(* IEC 61131-3 sources: BLM_BACKGROUND/src/PROGRAM_FILES/FC (part 5) *)

		General_State#STATE_END:
			CURRENT_STATE:=GENERAL_STATE#STATE_INIT;

	END_CASE;
	OutputState:=CURRENT_STATE;
END_FUNCTION_BLOCK

FUNCTION Init_Disp

  VAR_EXTERNAL
    Disp                            :ARRAY[(FIRST_DEVICE)..(FIRST_DEVICE+_MAXDEVICES#MAXDEVICES-1)] OF Device;
  END_VAR

  VAR_EXTERNAL CONSTANT
    INTERMEDIATE                    :SINT;
    FIRST_DEVICE                    :INT;
    DISP_IN_V_C :SINT;	//17 - Dispositivo virtuale composto da più dispositivi reali
    DISP_IN_TT  :SINT;		//01 - TEMPO LAVORO - TEMPO RIPOSO   xxxxxxx0001
  END_VAR

  VAR_INPUT
    Ndisp  :INT;
  END_VAR
  Disp[NDisp].Stato:=INTERMEDIATE;
  Disp[NDisp].position:=(DISP[Ndisp].Limite_Lavoro-DISP[Ndisp].Limite_Riposo)/2;
  DISP[NDisp].In_Movimento:=FALSE;
  AbilitazioneDispositivi(Dispositivo:=NDisp, Stato:=TRUE);
 (* {
  #ifdef EMULAZIONE_INPUT
  }*)
		IF Disp[NDisp].TipoIn<>DISP_IN_V_C THEN
			Disp[NDisp].TipoIn:=DISP_IN_TT;
    END_IF;
	(*{
  #endif  //Fine EMULAZIONE_INPUT
  }*)
END_FUNCTION

FUNCTION AbilitazioneDispositivi

  VAR_EXTERNAL
    Disp                            :ARRAY[(FIRST_DEVICE)..(FIRST_DEVICE+_MAXDEVICES#MAXDEVICES-1)] OF Device;
  END_VAR

  VAR_EXTERNAL CONSTANT
    FIRST_DEVICE                    :INT;
  END_VAR

  VAR_INPUT
    Dispositivo    :INT;
    Stato      :BOOL;
  END_VAR
  Disp[Dispositivo].consenso_minus:=Stato;
  Disp[Dispositivo].consenso_plus:=Stato;
END_FUNCTION

FUNCTION StartTimerRisparmioEnergetico

  VAR_EXTERNAL
    MinuteSavingEnergy              :INT;
    StatusStandBy                   :BOOL;
    TimerSistema                :ARRAY[0..MAX_TIMER_SISTEMA-1] OF Timer;
  END_VAR

  VAR_EXTERNAL CONSTANT
    T_ENERGY_SAVING    	            :INT;
    MAX_TIMER_SISTEMA 	            :USINT;
  END_VAR

  VAR_INPUT
    Tempo  :INT;
  END_VAR;
  IF MinuteSavingEnergy>0 THEN
    StatusStandBy:=FALSE;
    TimerSistema[T_ENERGY_SAVING].Value:=Tempo*60000.0;
    TimerSistema[T_ENERGY_SAVING].Status:=SINT#1;
  END_IF;
END_FUNCTION

FUNCTION ReadDigitalInput:BOOL

  VAR_EXTERNAL
    SystemStarted                   :BOOL;
    IAddress                        : ARRAY [0..MAXDIGITALINPUT] OF Digital_Input;
    O_EmergencyFromSimotion		      :BOOL;	//Only to be able to compile machines without safety PLCs
    InputWithoutAddress             :DINT;
    i_sys_DpCoupler                 :BOOL;
    i_sys_PnCoupler                 :BOOL;
    i_sys_StatusIOoptional          :BOOL;
    i_sys_StatusIOAL42               :BOOL;
    i_sys_StatusIOAL5                :BOOL;
    i_sys_StatusIOAL5Optional       :BOOL;
  END_VAR

  VAR_EXTERNAL CONSTANT
    MAXDIGITALINPUT                    :INT;
    INP_OUT_TIPO_SAFETY					       :SINT;
    INP_EMERGENCY                      :INT;
    ERR_IO_NOT_DEFINED                 :DINT ; //Manca associazione virtuale/fisico
  END_VAR

  VAR_INPUT
    NumInput  :DINT;
    Verifica  :BOOL:=FALSE;
  END_VAR

  VAR
    Porta     :DINT;
    Bit       :USINT;
    iret      :INT;
    OldStato  :BOOL;
  END_VAR

  IF NumInput>=0 AND SystemStarted=TRUE THEN
    IF IAddress[NumInput].Enable_Forzatura=TRUE THEN
      (*{
      #ifdef EMULAZIONE
			}*)
				IF IAddress[NumInput].Stato_Forzatura=FALSE THEN
					ReadDigitalInput:=FALSE;
				ELSE
					ReadDigitalInput:=TRUE;
				END_IF;
      (*{
      #else  //Fine EMULAZIONE
      }*)
				IF IAddress[NumInput].Port=INP_OUT_TIPO_SAFETY OR IAddress[NumInput].Bit=INP_OUT_TIPO_SAFETY THEN
					//Gli ingressi il cui stato è impostato dal plc di sicurezza non si possono forzare, tranne
					//l^ingresso di emergenza che può essere forzato solo basso (per esigenze di teleassistenza).
					IF NumInput=INP_EMERGENCY AND IAddress[NumInput].Enable_Forzatura=TRUE THEN
						IAddress[NumInput].Stato_Forzatura:=FALSE;
						ReadDigitalInput:=FALSE;
						O_EmergencyFromSimotion:=TRUE;
					ELSE
          	IAddress[NumInput].Enable_Forzatura:=FALSE;
					END_IF;
        ELSE
					//Ingressi standard si possono forzare
          IF IAddress[NumInput].STATO_FORZATURA=FALSE THEN
            ReadDigitalInput:=FALSE;
          ELSE
            ReadDigitalInput:=TRUE;
          END_IF;
        END_IF;
      (*{
      #endif  //Fine NO EMULAZIONE
      }*)
    ELSE
      Porta:=IAddress[NumInput].Port;
      Bit:=TO_USINT(IAddress[NumInput].Bit);
      IF IAddress[NumInput].Port=INP_OUT_TIPO_SAFETY AND IAddress[NumInput].Bit=INP_OUT_TIPO_SAFETY THEN
        //Lettura dello stato degli ingressi che vengono valorizzati da informazioni proveniente dal plc di sicurezza
        ReadDigitalInput:=LetturaIngressiSafety(NumeroInput:=NumInput);
      ELSE
        //Lettura ingressi collegati ai moduli standard e non impostati dal plc di sicurezza
        IF Verifica=TRUE AND (Porta<0 OR Bit<0) THEN
          //Verifica, se necessario, la definizione del collegamento virtuale fisico
          InputWithoutAddress:=NumInput;
          iret:=Push_error(Code:=ERR_IO_NOT_DEFINED, Arresto:=FALSE);
          ReadDigitalInput:=FALSE;
        ELSE
          OldStato:=FALSE;
          ReadDigitalInput:=LetturaIngressiDpCoupler(OldStato:=OldStato,
                                                     UsoDpCoupler:=i_sys_DpCoupler,
                                                     Porta:=porta,
                                                     Bit:=bit);
          OldStato:=ReadDigitalInput;
          ReadDigitalInput:=LetturaIngressiPnCoupler(OldStato:=OldStato,
                                                     UsoPnCoupler:=i_sys_PnCoupler,
                                                     Porta:=porta,
                                                     Bit:=bit);
          OldStato:=ReadDigitalInput;
          ReadDigitalInput:=LetturaIngressiSiemensProfinet(OldStato:=OldStato,
                                                           Porta:=porta,
                                                           Bit:=bit);
          OldStato:=ReadDigitalInput;
          ReadDigitalInput:=LetturaIngressiSiemensProfibus(OldStato:=OldStato,
                                                           Porta:=porta,
                                                           Bit:=bit,
                                                           StatoIOopzionale:=i_sys_StatusIOoptional,
                                                           StatoIOAL42:=i_sys_StatusIOAL42,
                                                           StatoIOAL5:=i_sys_StatusIOAL5,
                                                           StatoIOAL5Opzionale:=i_sys_StatusIOAL5Optional);
          OldStato:=ReadDigitalInput;
          ReadDigitalInput:=LetturaIngressiFestoProfinet(OldStato:=OldStato,
                                                         Porta:=porta,
                                                         Bit:=bit);
        END_IF;
      END_IF;
      IF IAddress[NumInput].inversione=TRUE THEN
        ///Inversione dello stato dell^ingresso fisico se prevista la proprietà
        IF ReadDigitalInput=TRUE THEN
          ReadDigitalInput:=FALSE;
        ELSE
          ReadDigitalInput:=TRUE;
        END_IF;
      END_IF;
    END_IF;  //Fine else degli ingressi di tipo standard port>-1 bit>-1
  ELSE
    ReadDigitalInput:=FALSE;
  END_IF;
END_FUNCTION

/**************************************************
 * READING STATUS OF VALUED INPUTS VIA SAFETY PLC *
 **************************************************/

FUNCTION LetturaIngressiSafety:BOOL

  VAR_EXTERNAL
    I_Emergenza,
    I_Barriera,
    I_RiarmoAzionamenti,
    I_Barriera_2,
    I_Pedale,
    I_Hold_To_Run,
    I_Radar_Zona_1,
    I_Radar_Zona_2,
    I_Radar_Zona_3,
    //Stato degli ingressi dei moduli di sicurezza
        //Stato degli ingressi dei moduli di sicurezza
    I_Modulo_1_Input_1,I_Modulo_1_Input_2,I_Modulo_1_Input_3,I_Modulo_1_Input_4,
    I_Modulo_2_Input_1,I_Modulo_2_Input_2,I_Modulo_2_Input_3,I_Modulo_2_Input_4,
    I_Modulo_3_Input_1,I_Modulo_3_Input_2,I_Modulo_3_Input_3,I_Modulo_3_Input_4  : BOOL;
  END_VAR

  VAR_EXTERNAL CONSTANT
    INP_PHOTOCELLS_NOT_VIOLATED             :INT;
    INP_MEASURE_TERMINAL_TUBE               :INT;
    INP_SEARCH_WELD                         :INT;
    INP_INTEGRATED_SOUL                     :INT;
    INP_EMERGENCY                           :INT;
    INP_RESET_DRIVES                        :INT;
    INP_BARRIER_2                           :INT;
    INP_PEDALE_SAFETY                       :INT;
    INP_HOLD_TO_RUN                         :INT;
    INP_EMERGENCY_PLC_SAFETY						    :INT;
    INP_PHOTOCELLS_NOT_VIOLATED_PLC_SAFETY	:INT;
    INP_HOLD_TO_RUN_PLC_SAFETY						  :INT;
    INP_PEDALE_SAFETY_PLC_SAFETY					  :INT;
    INP_RESET_DRIVE_PLC_SAFETY				      :INT;
    INP_BARRIER_2_PLC_SAFETY						    :INT;
    INP_OPTICAL_REARMING_PLC_SAFETY					:INT;
    INP_BARRIERA_3_PLC_SAFETY						    :INT;
    INP_EMERGENCY_EXTERIOR_PLC_SAFETY				:INT;
    INP_EXTERNAL_BARRIER_PLC_SAFETY					:INT;
    INP_RESET_EXTERNAL_DRIVES_PLC_SAFETY	  :INT;
    INP_RADAR_ZONA_BIT_0_PLC_SAFETY					:INT;
    INP_RADAR_ZONA_BIT_1_PLC_SAFETY					:INT;
    INP_RADAR_ZONA_1                        :INT;
    INP_RADAR_ZONA_2                        :INT;
    INP_RADAR_ZONA_3                        :INT;
    INP_RADAR_ZONA_BIT_0                    :INT;
    INP_RADAR_ZONA_BIT_1                    :INT;

  END_VAR

  VAR_INPUT
    MeasuringInput         : DB_ANY;
    NumeroInput  :DINT;
  END_VAR

  VAR
    Weld_Marker : REF_TO TO_MeasuringInput;
  END_VAR

  CASE NumeroInput OF
    (*{
    #ifdef SAFETY_INTEGRATED
    }
      INP_SAFETY_UOMO_MORTO:
        LetturaIngressiSafety:=i_sys_UomoMorto;
    {
    #endif  //Fine SAFETY_INTEGRATED
    }*)
    (*{
    #ifdef ORBITALE
    }
      {
      #ifdef FOTOCELLULA_MISURA_X1 %%%%
      }*)
        // INP_MEASURE_TERMINAL_TUBE:
        //   IF _to.FotocellulaMisuraX1.actualinputstate=POSITIVE THEN
        //     LetturaIngressiSafety:=TRUE;
        //   ELSE
        //     LetturaIngressiSafety:=FALSE;
        //   END_IF;
      (*{
      #endif  //Fine FOTOCELLULA_MISURA_X1
      }
    {
    #else  //Fine ORBITALE
    }*)
      INP_SEARCH_WELD, INP_INTEGRATED_SOUL:
        //Nelle macchine prima serie si usava lo stesso ingresso fisico
        //per leggere due diversi dispositivi
        Weld_Marker:= AsMeasuringInputRef(MeasuringInput);
        IF Weld_Marker^.InputState = TRUE THEN
          LetturaIngressiSafety:=TRUE;
        ELSE
          LetturaIngressiSafety:=FALSE;
        END_IF;
    (*{
    #endif  //Fine NO ORBITALE
    }
    {
    #ifdef PROFINET
    }*)
      INP_EMERGENCY:
        LetturaIngressiSafety:=I_Emergenza;
      INP_PHOTOCELLS_NOT_VIOLATED:
        LetturaIngressiSafety:=I_Barriera;
        INP_RESET_DRIVES:
        LetturaIngressiSafety:=I_RiarmoAzionamenti;
      INP_BARRIER_2:
        LetturaIngressiSafety:=I_Barriera_2;
			(*{
      #ifndef ORBITALE
      }*)
        INP_PEDALE_SAFETY:
          LetturaIngressiSafety:=I_Pedale;
        INP_HOLD_TO_RUN:
          LetturaIngressiSafety:=I_Hold_To_Run;
      (*{
      #endif  //Fine NO ORBITALE
      }
			{
			#ifdef DIAGNOSTICA_PLC_SAFETY
			}*)
				//Ingressi di diagnosdtica per visualizzazione in BlmMotion
				INP_EMERGENCY_PLC_SAFETY:
					LetturaIngressiSafety:=I_Modulo_1_Input_1;
        INP_PHOTOCELLS_NOT_VIOLATED_PLC_SAFETY:
					LetturaIngressiSafety:=I_Modulo_1_Input_2;
				(*{
				#ifndef ORBITALE
				}*)
					INP_HOLD_TO_RUN_PLC_SAFETY:
						LetturaIngressiSafety:=I_Modulo_1_Input_3;
					INP_PEDALE_SAFETY_PLC_SAFETY:
						LetturaIngressiSafety:=I_Modulo_2_Input_1;
				(*{
				#endif	//Fine NO ORBITALE
				}*)
				INP_RESET_DRIVE_PLC_SAFETY:
					LetturaIngressiSafety:=I_Modulo_1_Input_4;
				(*{
				#ifdef PLC_S7_1500
				}*)
					//Nuovo hardware associato a Tia portal
					INP_BARRIER_2_PLC_SAFETY:
						LetturaIngressiSafety:=I_Modulo_2_Input_2;
          INP_OPTICAL_REARMING_PLC_SAFETY	:
						LetturaIngressiSafety:=I_Modulo_2_Input_3;
					INP_BARRIERA_3_PLC_SAFETY:
						LetturaIngressiSafety:=I_Modulo_2_Input_4;
          INP_EMERGENCY_EXTERIOR_PLC_SAFETY:
						LetturaIngressiSafety:=I_Modulo_3_Input_1;
          INP_EXTERNAL_BARRIER_PLC_SAFETY:
						LetturaIngressiSafety:=I_Modulo_3_Input_2;
          INP_RESET_EXTERNAL_DRIVES_PLC_SAFETY:
						LetturaIngressiSafety:=I_Modulo_3_Input_3;
				(*{
				#else //FINE PLC_S7_1500
				}*)
					//Vecchio hardware associato a Step7
					(*{
					#ifdef ORBITALE
					}
            INP_BARRIER_2_PLC_SAFETY:
							(*{
							#ifdef DH4010
							}
								LetturaIngressiSafety:=I_Modulo_2_Input_2;
							(*{
							#else	//Fine DH4010
							}
								LetturaIngressiSafety:=I_Modulo_1_Input_3;
							(*{
							#endif	//Fine NO DH4010
							}
					{
					#else	//Fine ORBITALE
					}
            INP_BARRIER_2_PLC_SAFETY:
							LetturaIngressiSafety:=I_Modulo_2_Input_2;*)
						INP_RADAR_ZONA_BIT_0_PLC_SAFETY:
							LetturaIngressiSafety:=I_Modulo_2_Input_3;
						INP_RADAR_ZONA_BIT_1_PLC_SAFETY:
							LetturaIngressiSafety:=I_Modulo_2_Input_4;
						//Con la selezione a 3 bit di 3 zone radar l^impostazione
						//degli ingressi che vengono realmente cablati al PLC safety è:
						//0 0 1 = Zona 1
						//0 1 0 = Zona 2
						//1 0 0 = Zona 3
						INP_RADAR_ZONA_1:
							LetturaIngressiSafety:=I_Radar_Zona_1;
						INP_RADAR_ZONA_2:
							LetturaIngressiSafety:=I_Radar_Zona_2;
						INP_RADAR_ZONA_3:
							LetturaIngressiSafety:=I_Radar_Zona_3;
						//Con la selezione a 2 bit di 3 zone l^impostazione
						//degli ingressi che vengono realmente cablati al PLC safety è:
						//1 0 = Zona 1
						//0 1 = Zona 2
						//0 0 = Zona 3
						INP_RADAR_ZONA_BIT_0:
							IF I_Radar_Zona_1=TRUE THEN
								LetturaIngressiSafety:=FALSE;
							END_IF;
							IF I_Radar_Zona_2=TRUE THEN
								LetturaIngressiSafety:=TRUE;
							END_IF;
							IF I_Radar_Zona_3=TRUE THEN
								LetturaIngressiSafety:=FALSE;
							END_IF;
						INP_RADAR_ZONA_BIT_1:
							IF I_Radar_Zona_1=TRUE THEN
								LetturaIngressiSafety:=TRUE;
							END_IF;
							IF I_Radar_Zona_2=TRUE THEN
								LetturaIngressiSafety:=FALSE;
							END_IF;
							IF I_Radar_Zona_3=TRUE THEN
								LetturaIngressiSafety:=FALSE;
							END_IF;
					(*{
					#endif	//Fine NO ORBITALE
					}
				{
				#endif //FINE NO PLC_S7_1500
				}
			{
			#endif	//Fine DIAGNOSTICA_PLC_SAFETY
			}
    {
    #endif  //Fine PROFINET
    } *)
  END_CASE;
END_FUNCTION

FUNCTION LetturaIngressiDpCoupler:BOOL

  VAR_EXTERNAL
    V_dbcoupler_i  : dbcoupler_i;
  END_VAR

  VAR_INPUT
    OldStato      :BOOL;
    UsoDpCoupler  :BOOL;
    Porta					:DINT;
    Bit						:USINT;
  END_VAR

    LetturaIngressiDpCoupler:=OldStato;
    IF UsoDpCoupler=TRUE THEN
      CASE porta OF
      //Ingressi da DpCoupler
      900:LetturaIngressiDpCoupler:=getbit(V_dbcoupler_i.address_db_i[0], bit);//dbcoupler_i00.%X0; //_getbit(dbcoupler_i00, bit);
      901:LetturaIngressiDpCoupler:=getbit(V_dbcoupler_i.address_db_i[1], bit);
      902:LetturaIngressiDpCoupler:=getbit(V_dbcoupler_i.address_db_i[2], bit);
      903:LetturaIngressiDpCoupler:=getbit(V_dbcoupler_i.address_db_i[3], bit);
      904:LetturaIngressiDpCoupler:=getbit(V_dbcoupler_i.address_db_i[4], bit);
      905:LetturaIngressiDpCoupler:=getbit(V_dbcoupler_i.address_db_i[5], bit);
      906:LetturaIngressiDpCoupler:=getbit(V_dbcoupler_i.address_db_i[6], bit);
      907:LetturaIngressiDpCoupler:=getbit(V_dbcoupler_i.address_db_i[7], bit);
      908:LetturaIngressiDpCoupler:=getbit(V_dbcoupler_i.address_db_i[8], bit);
      909:LetturaIngressiDpCoupler:=getbit(V_dbcoupler_i.address_db_i[9], bit);
      910:LetturaIngressiDpCoupler:=getbit(V_dbcoupler_i.address_db_i[10], bit);
      911:LetturaIngressiDpCoupler:=getbit(V_dbcoupler_i.address_db_i[11], bit);
      912:LetturaIngressiDpCoupler:=getbit(V_dbcoupler_i.address_db_i[12], bit);
      913:LetturaIngressiDpCoupler:=getbit(V_dbcoupler_i.address_db_i[13], bit);
      914:LetturaIngressiDpCoupler:=getbit(V_dbcoupler_i.address_db_i[14], bit);
      915:LetturaIngressiDpCoupler:=getbit(V_dbcoupler_i.address_db_i[15], bit);
      916:LetturaIngressiDpCoupler:=getbit(V_dbcoupler_i.address_db_i[16], bit);
      917:LetturaIngressiDpCoupler:=getbit(V_dbcoupler_i.address_db_i[17], bit);
      918:LetturaIngressiDpCoupler:=getbit(V_dbcoupler_i.address_db_i[18], bit);
      919:LetturaIngressiDpCoupler:=getbit(V_dbcoupler_i.address_db_i[19], bit);
      920:LetturaIngressiDpCoupler:=getbit(V_dbcoupler_i.address_db_i[20], bit);
      921:LetturaIngressiDpCoupler:=getbit(V_dbcoupler_i.address_db_i[21], bit);
      922:LetturaIngressiDpCoupler:=getbit(V_dbcoupler_i.address_db_i[22], bit);
      923:LetturaIngressiDpCoupler:=getbit(V_dbcoupler_i.address_db_i[23], bit);
      924:LetturaIngressiDpCoupler:=getbit(V_dbcoupler_i.address_db_i[24], bit);
      925:LetturaIngressiDpCoupler:=getbit(V_dbcoupler_i.address_db_i[25], bit);
      926:LetturaIngressiDpCoupler:=getbit(V_dbcoupler_i.address_db_i[26], bit);
      927:LetturaIngressiDpCoupler:=getbit(V_dbcoupler_i.address_db_i[27], bit);
      928:LetturaIngressiDpCoupler:=getbit(V_dbcoupler_i.address_db_i[28], bit);
      929:LetturaIngressiDpCoupler:=getbit(V_dbcoupler_i.address_db_i[29], bit);
      930:LetturaIngressiDpCoupler:=getbit(V_dbcoupler_i.address_db_i[30], bit);
      931:LetturaIngressiDpCoupler:=getbit(V_dbcoupler_i.address_db_i[31], bit);
      932:LetturaIngressiDpCoupler:=getbit(V_dbcoupler_i.address_db_i[32], bit);
      933:LetturaIngressiDpCoupler:=getbit(V_dbcoupler_i.address_db_i[33], bit);
      934:LetturaIngressiDpCoupler:=getbit(V_dbcoupler_i.address_db_i[34], bit);
      935:LetturaIngressiDpCoupler:=getbit(V_dbcoupler_i.address_db_i[35], bit);
      936:LetturaIngressiDpCoupler:=getbit(V_dbcoupler_i.address_db_i[36], bit);
      937:LetturaIngressiDpCoupler:=getbit(V_dbcoupler_i.address_db_i[37], bit);
      938:LetturaIngressiDpCoupler:=getbit(V_dbcoupler_i.address_db_i[38], bit);
      939:LetturaIngressiDpCoupler:=getbit(V_dbcoupler_i.address_db_i[39], bit);
      940:LetturaIngressiDpCoupler:=getbit(V_dbcoupler_i.address_db_i[40], bit);
      941:LetturaIngressiDpCoupler:=getbit(V_dbcoupler_i.address_db_i[41], bit);
      942:LetturaIngressiDpCoupler:=getbit(V_dbcoupler_i.address_db_i[42], bit);
      943:LetturaIngressiDpCoupler:=getbit(V_dbcoupler_i.address_db_i[43], bit);
      944:LetturaIngressiDpCoupler:=getbit(V_dbcoupler_i.address_db_i[44], bit);
      945:LetturaIngressiDpCoupler:=getbit(V_dbcoupler_i.address_db_i[45], bit);
      946:LetturaIngressiDpCoupler:=getbit(V_dbcoupler_i.address_db_i[46], bit);
      947:LetturaIngressiDpCoupler:=getbit(V_dbcoupler_i.address_db_i[47], bit);
      948:LetturaIngressiDpCoupler:=getbit(V_dbcoupler_i.address_db_i[48], bit);
      949:LetturaIngressiDpCoupler:=getbit(V_dbcoupler_i.address_db_i[49], bit);
      950:LetturaIngressiDpCoupler:=getbit(V_dbcoupler_i.address_db_i[50], bit);
      951:LetturaIngressiDpCoupler:=getbit(V_dbcoupler_i.address_db_i[51], bit);
      952:LetturaIngressiDpCoupler:=getbit(V_dbcoupler_i.address_db_i[52], bit);
      953:LetturaIngressiDpCoupler:=getbit(V_dbcoupler_i.address_db_i[53], bit);
      954:LetturaIngressiDpCoupler:=getbit(V_dbcoupler_i.address_db_i[54], bit);
      955:LetturaIngressiDpCoupler:=getbit(V_dbcoupler_i.address_db_i[55], bit);
      956:LetturaIngressiDpCoupler:=getbit(V_dbcoupler_i.address_db_i[56], bit);
      957:LetturaIngressiDpCoupler:=getbit(V_dbcoupler_i.address_db_i[57], bit);
      958:LetturaIngressiDpCoupler:=getbit(V_dbcoupler_i.address_db_i[58], bit);
      959:LetturaIngressiDpCoupler:=getbit(V_dbcoupler_i.address_db_i[59], bit);
      960:LetturaIngressiDpCoupler:=getbit(V_dbcoupler_i.address_db_i[60], bit);
      961:LetturaIngressiDpCoupler:=getbit(V_dbcoupler_i.address_db_i[61], bit);
      962:LetturaIngressiDpCoupler:=getbit(V_dbcoupler_i.address_db_i[62], bit);
      963:LetturaIngressiDpCoupler:=getbit(V_dbcoupler_i.address_db_i[63], bit);
    END_CASE;
  END_IF;
END_FUNCTION

/***********************************************************************
 * READING STATUS OF VALUED INPUTS VIA PNPNCOUPLER ON PROFINET NETWORK *
 ***********************************************************************/

 FUNCTION LetturaIngressiPnCoupler:BOOL

  VAR_EXTERNAL
    V_pncoupler_i  : pncoupler_i;

  END_VAR

  VAR_INPUT
    OldStato      :BOOL;
    UsoPnCoupler	:BOOL;
    Porta					:DINT;
    Bit						:USINT;
  END_VAR
  LetturaIngressiPnCoupler:=OldStato;
  {::ifdef PROFINET}
    IF UsoPnCoupler=TRUE THEN
      CASE porta OF
        //Ingressi da PnCoupler
        900:LetturaIngressiPnCoupler:=getbit(V_pncoupler_i.address_pn_i[0], bit);
        901:LetturaIngressiPnCoupler:=getbit(V_pncoupler_i.address_pn_i[1], bit);
        902:LetturaIngressiPnCoupler:=getbit(V_pncoupler_i.address_pn_i[2], bit);
        903:LetturaIngressiPnCoupler:=getbit(V_pncoupler_i.address_pn_i[3], bit);
        904:LetturaIngressiPnCoupler:=getbit(V_pncoupler_i.address_pn_i[4], bit);
        905:LetturaIngressiPnCoupler:=getbit(V_pncoupler_i.address_pn_i[5], bit);
        906:LetturaIngressiPnCoupler:=getbit(V_pncoupler_i.address_pn_i[6], bit);
        907:LetturaIngressiPnCoupler:=getbit(V_pncoupler_i.address_pn_i[7], bit);
        908:LetturaIngressiPnCoupler:=getbit(V_pncoupler_i.address_pn_i[8], bit);
        909:LetturaIngressiPnCoupler:=getbit(V_pncoupler_i.address_pn_i[9], bit);
        910:LetturaIngressiPnCoupler:=getbit(V_pncoupler_i.address_pn_i[10], bit);
        911:LetturaIngressiPnCoupler:=getbit(V_pncoupler_i.address_pn_i[11], bit);
        912:LetturaIngressiPnCoupler:=getbit(V_pncoupler_i.address_pn_i[12], bit);
        913:LetturaIngressiPnCoupler:=getbit(V_pncoupler_i.address_pn_i[13], bit);
        914:LetturaIngressiPnCoupler:=getbit(V_pncoupler_i.address_pn_i[14], bit);
        915:LetturaIngressiPnCoupler:=getbit(V_pncoupler_i.address_pn_i[15], bit);
        916:LetturaIngressiPnCoupler:=getbit(V_pncoupler_i.address_pn_i[16], bit);
        917:LetturaIngressiPnCoupler:=getbit(V_pncoupler_i.address_pn_i[17], bit);
        918:LetturaIngressiPnCoupler:=getbit(V_pncoupler_i.address_pn_i[18], bit);
        919:LetturaIngressiPnCoupler:=getbit(V_pncoupler_i.address_pn_i[19], bit);
        920:LetturaIngressiPnCoupler:=getbit(V_pncoupler_i.address_pn_i[20], bit);
        921:LetturaIngressiPnCoupler:=getbit(V_pncoupler_i.address_pn_i[21], bit);
        922:LetturaIngressiPnCoupler:=getbit(V_pncoupler_i.address_pn_i[22], bit);
        923:LetturaIngressiPnCoupler:=getbit(V_pncoupler_i.address_pn_i[23], bit);
        924:LetturaIngressiPnCoupler:=getbit(V_pncoupler_i.address_pn_i[23], bit);
        925:LetturaIngressiPnCoupler:=getbit(V_pncoupler_i.address_pn_i[25], bit);
        926:LetturaIngressiPnCoupler:=getbit(V_pncoupler_i.address_pn_i[26], bit);
        927:LetturaIngressiPnCoupler:=getbit(V_pncoupler_i.address_pn_i[27], bit);
        928:LetturaIngressiPnCoupler:=getbit(V_pncoupler_i.address_pn_i[28], bit);
        929:LetturaIngressiPnCoupler:=getbit(V_pncoupler_i.address_pn_i[29], bit);
        930:LetturaIngressiPnCoupler:=getbit(V_pncoupler_i.address_pn_i[30], bit);
        931:LetturaIngressiPnCoupler:=getbit(V_pncoupler_i.address_pn_i[31], bit);
        932:LetturaIngressiPnCoupler:=getbit(V_pncoupler_i.address_pn_i[32], bit);
        933:LetturaIngressiPnCoupler:=getbit(V_pncoupler_i.address_pn_i[33], bit);
        934:LetturaIngressiPnCoupler:=getbit(V_pncoupler_i.address_pn_i[34], bit);
        935:LetturaIngressiPnCoupler:=getbit(V_pncoupler_i.address_pn_i[35], bit);
        936:LetturaIngressiPnCoupler:=getbit(V_pncoupler_i.address_pn_i[36], bit);
        937:LetturaIngressiPnCoupler:=getbit(V_pncoupler_i.address_pn_i[37], bit);
        938:LetturaIngressiPnCoupler:=getbit(V_pncoupler_i.address_pn_i[38], bit);
        939:LetturaIngressiPnCoupler:=getbit(V_pncoupler_i.address_pn_i[39], bit);
        940:LetturaIngressiPnCoupler:=getbit(V_pncoupler_i.address_pn_i[40], bit);
        941:LetturaIngressiPnCoupler:=getbit(V_pncoupler_i.address_pn_i[41], bit);
        942:LetturaIngressiPnCoupler:=getbit(V_pncoupler_i.address_pn_i[42], bit);
        943:LetturaIngressiPnCoupler:=getbit(V_pncoupler_i.address_pn_i[43], bit);
        944:LetturaIngressiPnCoupler:=getbit(V_pncoupler_i.address_pn_i[44], bit);
        945:LetturaIngressiPnCoupler:=getbit(V_pncoupler_i.address_pn_i[45], bit);
        946:LetturaIngressiPnCoupler:=getbit(V_pncoupler_i.address_pn_i[46], bit);
        947:LetturaIngressiPnCoupler:=getbit(V_pncoupler_i.address_pn_i[47], bit);
        948:LetturaIngressiPnCoupler:=getbit(V_pncoupler_i.address_pn_i[48], bit);
        949:LetturaIngressiPnCoupler:=getbit(V_pncoupler_i.address_pn_i[49], bit);
        950:LetturaIngressiPnCoupler:=getbit(V_pncoupler_i.address_pn_i[50], bit);
        951:LetturaIngressiPnCoupler:=getbit(V_pncoupler_i.address_pn_i[51], bit);
        952:LetturaIngressiPnCoupler:=getbit(V_pncoupler_i.address_pn_i[52], bit);
        953:LetturaIngressiPnCoupler:=getbit(V_pncoupler_i.address_pn_i[53], bit);
        954:LetturaIngressiPnCoupler:=getbit(V_pncoupler_i.address_pn_i[54], bit);
        955:LetturaIngressiPnCoupler:=getbit(V_pncoupler_i.address_pn_i[55], bit);
        956:LetturaIngressiPnCoupler:=getbit(V_pncoupler_i.address_pn_i[56], bit);
        957:LetturaIngressiPnCoupler:=getbit(V_pncoupler_i.address_pn_i[57], bit);
        958:LetturaIngressiPnCoupler:=getbit(V_pncoupler_i.address_pn_i[58], bit);
        959:LetturaIngressiPnCoupler:=getbit(V_pncoupler_i.address_pn_i[59], bit);
        960:LetturaIngressiPnCoupler:=getbit(V_pncoupler_i.address_pn_i[60], bit);
        961:LetturaIngressiPnCoupler:=getbit(V_pncoupler_i.address_pn_i[61], bit);
        962:LetturaIngressiPnCoupler:=getbit(V_pncoupler_i.address_pn_i[62], bit);
        963:LetturaIngressiPnCoupler:=getbit(V_pncoupler_i.address_pn_i[63], bit);
      END_CASE;
    END_IF;
  {::endif}  //Fine PROFINET

END_FUNCTION

FUNCTION LetturaIngressiSiemensProfinet:BOOL

  VAR_EXTERNAL
    i_sys_StatoIOAL5_old			              :BOOL;
    i_sys_StatoIOAL5Opzionale_old           :BOOL;
    i_sys_StatoIOAL5                        :BOOL;
    i_sys_StatoIOAL5Opzionale               :BOOL;
    V_ph_i  : ph_i;
    V_ph_i_old  : ph_i_old;
    V_PHIAL5_Opz  : PHIAL5_Opz;
    V_PHIAL5_Opz_old  : PHIAL5_Opz_old;

                X122_d0 : BOOL;
                X122_d1 : BOOL;
                X122_d2 : BOOL;
                X122_d3 : BOOL;
                X122_d16 : BOOL;
                X122_d17 : BOOL;

                X132_d4 : BOOL;
                X132_d5 : BOOL;
                X132_d6 : BOOL;
                X132_d7 : BOOL;
                X132_d20 : BOOL;
                X132_d21 : BOOL;
  END_VAR

  VAR_EXTERNAL CONSTANT
    INDIRIZZO_X122_SINAMICS             :INT;
    INDIRIZZO_X132_SINAMICS             :INT;
  END_VAR

  VAR_INPUT
    OldStato:BOOL;
    Porta		:DINT;
    Bit			:USINT;
  END_VAR;

  LetturaIngressiSiemensProfinet:=OldStato;
  CASE Porta OF
    //Macchine seconda serie con profinet
    00:LetturaIngressiSiemensProfinet:=getbit(V_ph_i.address_ph_i[0], bit);  //32.0÷7
    01:LetturaIngressiSiemensProfinet:=getbit(V_ph_i.address_ph_i[1], bit);  //33.0÷7
    02:LetturaIngressiSiemensProfinet:=getbit(V_ph_i.address_ph_i[2], bit);  //34.0÷7
    //Ingressi opzionali
    03:LetturaIngressiSiemensProfinet:=getbit(V_ph_i.address_ph_i[3], bit);  //37.0÷7
    04:LetturaIngressiSiemensProfinet:=getbit(V_ph_i.address_ph_i[4], bit);  //38.0÷7
  END_CASE;
  {::ifdef AL_BLM}
    IF i_sys_StatoIOAL5_old=TRUE THEN
      CASE Porta OF
        //IM 151-3 PN ST (STEP 7)ingressi standard AL5
        08:LetturaIngressiSiemensProfinet:=getbit(V_ph_i_old.address_ph_i_old[0], bit);  //42.0÷3
        09:LetturaIngressiSiemensProfinet:=getbit(V_ph_i_old.address_ph_i_old[1], bit);  //43.0÷3
        10:LetturaIngressiSiemensProfinet:=getbit(V_ph_i_old.address_ph_i_old[2], bit);  //44.0÷3
        11:LetturaIngressiSiemensProfinet:=getbit(V_ph_i_old.address_ph_i_old[3], bit);  //45.0÷3
        12:LetturaIngressiSiemensProfinet:=getbit(V_ph_i_old.address_ph_i_old[4], bit);  //46.0÷3
        13:LetturaIngressiSiemensProfinet:=getbit(V_ph_i_old.address_ph_i_old[5], bit);  //47.0÷3
        14:LetturaIngressiSiemensProfinet:=getbit(V_ph_i_old.address_ph_i_old[6], bit);  //48.0÷3
      END_CASE;
    END_IF;
    IF i_sys_StatoIOAL5Opzionale_old=TRUE THEN
      CASE Porta OF
        //IM 151-3 PN ST (STEP 7)ingressi opzionali
        15:LetturaIngressiSiemensProfinet:=getbit(V_PHIAL5_Opz_old.address_PHIAL5_Opz_old[0], bit);  //49.0÷3
        16:LetturaIngressiSiemensProfinet:=getbit(V_PHIAL5_Opz_old.address_PHIAL5_Opz_old[1], bit);  //50.0÷3
        17:LetturaIngressiSiemensProfinet:=getbit(V_PHIAL5_Opz_old.address_PHIAL5_Opz_old[2], bit);  //51.0÷3
        18:LetturaIngressiSiemensProfinet:=getbit(V_PHIAL5_Opz_old.address_PHIAL5_Opz_old[3], bit);  //52.0÷3
        19:LetturaIngressiSiemensProfinet:=getbit(V_PHIAL5_Opz_old.address_PHIAL5_Opz_old[4], bit);  //53.0÷3
        20:LetturaIngressiSiemensProfinet:=getbit(V_PHIAL5_Opz_old.address_PHIAL5_Opz_old[5], bit);  //54.0÷3
        21:LetturaIngressiSiemensProfinet:=getbit(V_PHIAL5_Opz_old.address_PHIAL5_Opz_old[6], bit);  //55.0÷3
      END_CASE;
    END_IF;

    IF i_sys_StatoIOAL5=TRUE THEN
      //IM 155-6 PN HF (TIA PORTAL) ingressi standard AL5
      CASE Porta OF
        05:LetturaIngressiSiemensProfinet:=getbit(V_ph_i_old.address_ph_i_old[0], bit);  //42.0÷7
        06:LetturaIngressiSiemensProfinet:=getbit(V_ph_i_old.address_ph_i_old[1], bit);  //43.0÷7
        07:LetturaIngressiSiemensProfinet:=getbit(V_ph_i_old.address_ph_i_old[2], bit);  //44.0÷7
        08:LetturaIngressiSiemensProfinet:=getbit(V_ph_i_old.address_ph_i_old[3], bit);  //45.0÷7
      END_CASE;
    END_IF;
    IF i_sys_StatoIOAL5Opzionale THEN
      //IM 155-6 PN HF (TIA PORTAL) ingressi opzionali
      CASE Porta OF
        12:LetturaIngressiSiemensProfinet:=getbit(V_PHIAL5_Opz.address_PHIAL5_Opz[0], bit);  //49.0÷7
        13:LetturaIngressiSiemensProfinet:=getbit(V_PHIAL5_Opz.address_PHIAL5_Opz[1], bit);  //50.0÷7
        14:LetturaIngressiSiemensProfinet:=getbit(V_PHIAL5_Opz.address_PHIAL5_Opz[2], bit);  //51.0÷7
        15:LetturaIngressiSiemensProfinet:=getbit(V_PHIAL5_Opz.address_PHIAL5_Opz[3], bit);  //52.0÷7
      END_CASE;
    END_IF;
  {::endif}  //Fine AL_BLM

  // CASE Porta OF
    // {::ifdef TAVOLI_ELETTRICI} %%%%

    //   23:LetturaIngressiSiemensProfinet:=getbit(I_Tavoli_0, bit);
    //   24:LetturaIngressiSiemensProfinet:=getbit(I_Tavoli_1, bit);
    //   25:LetturaIngressiSiemensProfinet:=getbit(I_Tavoli_2, bit);
    // {::endif} //FINE TAVOLI ELETTRICI

      {::ifndef EMULAZIONE}

      INDIRIZZO_X122_SINAMICS:
        CASE bit OF
          0:LetturaIngressiSiemensProfinet:=X122_d0;
          1:LetturaIngressiSiemensProfinet:=X122_d1;
          2:LetturaIngressiSiemensProfinet:=X122_d2;
          3:LetturaIngressiSiemensProfinet:=X122_d3;
          8:LetturaIngressiSiemensProfinet:=X122_d16;
          9:LetturaIngressiSiemensProfinet:=X122_d17;
        END_CASE;

      INDIRIZZO_X132_SINAMICS:
        CASE bit OF
          0:LetturaIngressiSiemensProfinet:=X132_d4;
          1:LetturaIngressiSiemensProfinet:=X132_d5;
          2:LetturaIngressiSiemensProfinet:=X132_d6;
          3:LetturaIngressiSiemensProfinet:=X132_d7;
          8:LetturaIngressiSiemensProfinet:=X132_d20;
          9:LetturaIngressiSiemensProfinet:=X132_d21;
        END_CASE;
      {::endif}  //Fine NO EMULAZIONE

  // END_CASE;

END_FUNCTION
// {
// #else //FINE PLC_S7_1500
// }

/**************************************************************************
 * READING STATUS OF INPUTS VALUED BY SIEMENS MODULES ON PROFIBUS NETWORK *
 **************************************************************************/

FUNCTION LetturaIngressiSiemensProfibus:BOOL

  VAR_EXTERNAL
    X122_d0 : BOOL;
    X122_d1 : BOOL;
    X122_d2 : BOOL;
    X122_d3 : BOOL;

    X132_d4 : BOOL;
    X132_d5 : BOOL;
    X132_d6 : BOOL;
    X132_d7 : BOOL;

    V_ph_i                   : ph_i;
    V_PHIAL5_Opz             : PHIAL5_Opz;

    // PHIAL5_Opz_1  :BYTE;
    // PHIAL5_Opz_2 :BYTE;
    // PHIAL5_Opz_3 :BYTE;
    // PHIAL5_Opz_4 :BYTE;
    // PHIAL5_Opz_5  :BYTE;
    // PHIAL5_Opz_6 :BYTE;
    // PHIAL5_Opz_7  :BYTE;

    // phi00  :BYTE;
    // phi01  :BYTE;
    // phi02  :BYTE;
    // phi03  :BYTE;
    // phi04  :BYTE;
  END_VAR

  VAR_EXTERNAL CONSTANT
    INDIRIZZO_X122_SINAMICS             :INT;
    INDIRIZZO_X132_SINAMICS             :INT;
  END_VAR

  VAR_INPUT
    OldStato            :BOOL;
    Porta								:DINT;
    Bit									:USINT;
    StatoIOopzionale    :BOOL;
    StatoIOAL42					:BOOL;
    StatoIOAL5          :BOOL;
    StatoIOAL5Opzionale	:BOOL;
  END_VAR

  LetturaIngressiSiemensProfibus:=OldStato;
  //{::ifndef PROFINET}%%%%
    // IF StatoIOopzionale=TRUE THEN %%%%
      //Modulo IO opzionale
    //   CASE porta OF
    //     00:LetturaIngressiSiemensProfibus:=getbit(PHI00_opzionale,bit);
    //     01:LetturaIngressiSiemensProfibus:=getbit(PHI01_opzionale,bit);
    //     02:LetturaIngressiSiemensProfibus:=getbit(PHI02_opzionale,bit);
    //     03:LetturaIngressiSiemensProfibus:=getbit(PHI03_opzionale,bit);
    //     04:LetturaIngressiSiemensProfibus:=getbit(PHI04_opzionale,bit);
    //     08:LetturaIngressiSiemensProfibus:=getbit(PHI08_opzionale,bit);
    //     09:LetturaIngressiSiemensProfibus:=getbit(PHI09_opzionale,bit);
    //     10:LetturaIngressiSiemensProfibus:=getbit(PHI10_opzionale,bit);
    //   END_CASE;
    // ELSE
    //   //Modulo IO standard
    //   CASE porta OF
    //     00:LetturaIngressiSiemensProfibus:=getbit(PHI00,bit);
    //     01:LetturaIngressiSiemensProfibus:=getbit(PHI01,bit);
    //     02:LetturaIngressiSiemensProfibus:=getbit(PHI02,bit);
    //     03:LetturaIngressiSiemensProfibus:=getbit(PHI03,bit);
    //     04:LetturaIngressiSiemensProfibus:=getbit(PHI04,bit);
    //   END_CASE;
    // END_IF;
    {::ifndef EMULAZIONE}
      CASE porta OF
        INDIRIZZO_X122_SINAMICS:
          CASE bit OF
            0:LetturaIngressiSiemensProfibus:=X122_d0;
            1:LetturaIngressiSiemensProfibus:=X122_d1;
            2:LetturaIngressiSiemensProfibus:=X122_d2;
            3:LetturaIngressiSiemensProfibus:=X122_d3;
          END_CASE;
        INDIRIZZO_X132_SINAMICS:
          CASE bit OF
            0:LetturaIngressiSiemensProfibus:=X132_d4;
            1:LetturaIngressiSiemensProfibus:=X132_d5;
            2:LetturaIngressiSiemensProfibus:=X132_d6;
            3:LetturaIngressiSiemensProfibus:=X132_d7;
          END_CASE;
      END_CASE;
    {::endif}  //Fine NO EMULAZIONE
    {::ifdef AL_BLM}
    //   {
    //   #ifdef ETURN %%%%
    //   }
        // IF StatoIOAL42=TRUE THEN
        //   CASE porta OF
        //     11:LetturaIngressiSiemensProfibus:=getbit(PHI20,bit);
        //     12:LetturaIngressiSiemensProfibus:=getbit(PHI21,bit);
        //     13:LetturaIngressiSiemensProfibus:=getbit(PHI22,bit);
        //     14:LetturaIngressiSiemensProfibus:=getbit(PHI23,bit);
        //     15:LetturaIngressiSiemensProfibus:=getbit(PHI24,bit);
        //   END_CASE;
        // END_IF;
      // {
      // #endif  //Fine ETURN
      // }
      // IF StatoIOAL5=TRUE THEN
      //   CASE porta OF
      //     11:LetturaIngressiSiemensProfibus:=getbit(PHI20_opzionale, bit);
      //     12:LetturaIngressiSiemensProfibus:=getbit(PHI21_opzionale, bit);
      //     13:LetturaIngressiSiemensProfibus:=getbit(PHI22_opzionale, bit);
      //     14:LetturaIngressiSiemensProfibus:=getbit(PHI23_opzionale, bit);
      //     15:LetturaIngressiSiemensProfibus:=getbit(PHI24_opzionale, bit);
      //     16:LetturaIngressiSiemensProfibus:=getbit(PHI25_opzionale, bit);
      //     17:LetturaIngressiSiemensProfibus:=getbit(PHI26_opzionale, bit);
      //   END_CASE;
      // END_IF;
      // {::ifdef MODULO_ROLAND} %%%%
      //   IF StatoIOAL5Opzionale=TRUE THEN
      //     CASE porta OF
      //       18:LetturaIngressiSiemensProfibus:=getbit(PHIAL5_Opz_1, bit);
      //       19:LetturaIngressiSiemensProfibus:=getbit(PHIAL5_Opz_2, bit);
      //       20:LetturaIngressiSiemensProfibus:=getbit(PHIAL5_Opz_3, bit);
      //       21:LetturaIngressiSiemensProfibus:=getbit(PHIAL5_Opz_4, bit);
      //       22:LetturaIngressiSiemensProfibus:=getbit(PHIAL5_Opz_5, bit);
      //       23:LetturaIngressiSiemensProfibus:=getbit(PHIAL5_Opz_6, bit);
      //       24:LetturaIngressiSiemensProfibus:=getbit(PHIAL5_Opz_7, bit);
      //     END_CASE;
      //   END_IF;
      // {::endif}  //Fine MODULO_ROLAND

  {::endif}  //Fine AL_BLM

  // {
  // #endif  //Fine NO PROFINET
  // }
END_FUNCTION

/**************************************************************************
 * READING STATUS OF INPUTS VALUED BY SIEMENS MODULES ON PROFIBUS NETWORK *
 **************************************************************************/

FUNCTION LetturaIngressiFestoProfinet:BOOL

  VAR_EXTERNAL CONSTANT
    FESTO_INP_LINEA_1_MODULO_1          :INT;  //bit 0÷15  16 input
    FESTO_INP_LINEA_1_MODULO_3          :INT;  //bit 0÷07  08 input
    FESTO_INP_LINEA_2_MODULO_2          :INT;  //bit 0÷15  16 input
    FESTO_INP_LINEA_2_MODULO_3          :INT;  //bit 0÷07  08 input
    FESTO_INP_LINEA_3_MODULO_2          :INT;  //bit 0÷15  16 input
    FESTO_INP_LINEA_3_MODULO_3          :INT;  //bit 0÷07  08 input
    FESTO_INP_LINEA_4_MODULO_2          :INT;  //bit 0÷15  16 input
    FESTO_INP_LINEA_4_MODULO_3          :INT;  //bit 0÷07  08 input
END_VAR

  VAR_INPUT
    OldStato	:BOOL;
    Porta			:DINT;
    Bit				:USINT;
  END_VAR
  LetturaIngressiFestoProfinet:=OldStato;
  {::ifdef IO_FESTO_PROFINET}
    CASE porta OF
      FESTO_INP_LINEA_1_MODULO_1:
        LetturaIngressiFestoProfinet:=getbit(festo_inp_linea_1a, bit);  //16 ingressi
      FESTO_INP_LINEA_1_MODULO_3:
        LetturaIngressiFestoProfinet:=getbit(festo_inp_linea_1b, bit);  //08 ingressi
      FESTO_INP_LINEA_2_MODULO_2:
        LetturaIngressiFestoProfinet:=getbit(festo_inp_linea_2a, bit);  //16 ingressi
      FESTO_INP_LINEA_2_MODULO_3:
        LetturaIngressiFestoProfinet:=getbit(festo_inp_linea_2b, bit);  //08 ingressi
      FESTO_INP_LINEA_3_MODULO_2:
        LetturaIngressiFestoProfinet:=getbit(festo_inp_linea_3a, bit);  //16 ingressi
      FESTO_INP_LINEA_3_MODULO_3:
        LetturaIngressiFestoProfinet:=getbit(festo_inp_linea_3b, bit);  //08 ingressi
      FESTO_INP_LINEA_4_MODULO_2:
        LetturaIngressiFestoProfinet:=getbit(festo_inp_linea_4a, bit);  //16 ingressi
      FESTO_INP_LINEA_4_MODULO_3:
        LetturaIngressiFestoProfinet:=getbit(festo_inp_linea_4b, bit);  //08 ingressi
    END_CASE;
  {::endif} //Fine IO_FESTO_PROFINET

  ;

END_FUNCTION

FUNCTION_BLOCK FB_EnableMasterAxisBLM

  VAR_EXTERNAL
    AssiMaster                      :ARRAY[FIRST_AXIS_MASTER..FIRST_AXIS_MASTER+_CONST_VAR_DEF._MAXAXIS_MASTER#MAXAXIS_MASTER-1] OF MasterAxis;
  END_VAR

  VAR_EXTERNAL CONSTANT

    FIRST_AXIS_MASTER				        :INT;

  END_VAR

	VAR_INPUT
		NumMaster	:INT;
		//Asse			:PosAxis;
	END_VAR

	VAR
		dret					:LREAL;
		CURRENT_STATE	:INT;
		//thisCommand		:CommandIDType;
	END_VAR

	VAR_OUTPUT
		OutputState:INT;
	END_VAR
	CASE CURRENT_STATE OF
		GENERAL_STATE#STATE_INIT:
			(*IF UsoPLCOpen THEN
				//PLCOpen*)
				AssiMaster[NumMaster].MC_Axes.enable_axes :=TRUE;
				CURRENT_STATE:=GENERAL_STATE#STATE_END;
			(*ELSE
				thisCommand:=_getCommandID();
				CURRENT_STATE:=STATE_ENABLEMASTER_ENABLE;
			END_IF;

		STATE_ENABLEMASTER_ENABLE:
			dret:=_enableAxis(axis:=Asse,
							movingMode:=POSITION_CONTROLLED,
							enableMode:=ALL,
							servoControlMode:=ACTIVE,
							servoCommandToActualMode:=INACTIVE,
							nextCommand:=IMMEDIATELY,
							commandId:=thisCommand,
							forcecontrolMode:=INACTIVE);
			IF (ModoAttesa=WHEN_COMMAND_DONE) THEN
				IF (dret<>7001 AND dret<>7002) THEN
					CURRENT_STATE:=STATE_END;
				END_IF;
			ELSE*)
				CURRENT_STATE:=GENERAL_STATE#STATE_END;
			//END_IF;

		GENERAL_STATE#STATE_END:
			CURRENT_STATE:=GENERAL_STATE#STATE_INIT;
	END_CASE;
	OutputState:=CURRENT_STATE;
END_FUNCTION_BLOCK

/**********************************************************************
 * RESET OF OUTPUTS THAT NEED TO BE RESET WITH CYCLE STOP AND STORAGE *
 *                     OF THE STATE BEFORE RESET                      *
 **********************************************************************/
FUNCTION OnStopCicloDispositivi

  VAR_EXTERNAL
    OAddress                        : ARRAY [0..MAXDIGITALOUTPUT] OF Digital_Output;
  END_VAR

  VAR_EXTERNAL CONSTANT
    MAXDIGITALOUTPUT                    :INT;
    MAXDIGITALINPUT                     :INT;
  END_VAR

  VAR
    i    :DINT;
  END_VAR;
  FOR i:=0 TO MAXDIGITALOUTPUT DO
    IF oaddress[i].AbilGestStopCiclo=TRUE THEN
			IF oaddress[i].stato=TRUE THEN
				//Si memorizza lo stato dell^uscita solamente se è attiva
				oaddress[i].statoprestopciclo:=oaddress[i].stato;
			END_IF;
      WriteDigitalOutput(NumOutput:=i, Value:=FALSE);
    END_IF;
  END_FOR;
END_FUNCTION

/*****************************************************************************
 * READS FROM THE STATE TABLE THE VALUE INDICATED BY THE ROW AND COLUMN. THE *
 *                 PROGRAMME NUMBER FROM 0 TO MAXPROGRAMS-1                  *
 *****************************************************************************/

FUNCTION ReadTabStati:REAL

  VAR_EXTERNAL
    Programmi                      :ARRAY[0.._CONST_VAR_DEF._MPROGRAMS#MAXPROGRAMS - UINT#1] OF Programma;
    // {
    // #ifdef DH4010
    // }
    TabellaStati	:ARRAY[TABLE#TABLE_LX ..TABLE#TABLE_RX ] OF TabStato;
  END_VAR

  VAR_EXTERNAL CONSTANT
    ERR_NUMSTATES                       :DINT;
  END_VAR

  VAR_INPUT
    Riga,
    Colonna,
    Programma	:INT;
    Tabella   :SINT;
  END_VAR

  VAR
    Puntatore	:DINT;
    iret      :INT;
  END_VAR

  ;
//  {
//   #ifdef DH4010
//   }
    // IF GetNumberOfStates(Tabella:=Tabella, Programma:=Programma)>0 THEN
    //   Puntatore:=Riga+Programmi[Programma].TabStatiInizio[Tabella];
    //   ReadTabStati:=TabellaStati[Tabella][Puntatore][Colonna];
    // ELSE
    //   iret:=Push_error(Code:=ERR_NUMSTATES, Arresto:=FALSE, Attesa:=FALSE);
    // END_IF;
  // {
  // #else  //Fine DH4010
  // }
    // IF GetNumberOfStates(Tabella:=Tabella, Programma:=Programma)>0 THEN
    //   Puntatore:=Riga+Programmi[Programma].TabStatiInizio;
    //   ReadTabStati:=TabellaStati[Puntatore][Colonna];
    // ELSE
    //   iret:=Push_error(Code:=ERR_NUMSTATES, Arresto:=FALSE, Attesa:=FALSE);
    // END_IF;
  // {
  // #endif  //Fine NO DH4010
  // }
END_FUNCTION

FUNCTION SetAxSwLimit1

  VAR_EXTERNAL
    pm                              : ARRAY[_FIRST_AXIS#FIRST_AXIS.._FIRST_AXIS#FIRST_AXIS+_CONST_VAR_DEF._MAXIS#MAXAXIS-1] OF AxisParameters;
  END_VAR

  VAR_EXTERNAL CONSTANT
    EXTRALIMIT         	:REAL ; // extralimite per limiti fisici
    Q1 : INT;
    V1 : INT;
  END_VAR

  VAR_INPUT
		PrimoAsseNoGestione		:INT:=-1;
		SecondoAsseNoGestione	:INT:=-1;
		TerzoAsseNoGestione		:INT:=-1;
		QuartoAsseNoGestione	:INT:=-1;
		QuintoAsseNoGestione	:INT:=-1;
		SestoAsseNoGestione		:INT:=-1;
  END_VAR
  VAR
    i											:INT;
		Eseguire							:BOOL:=TRUE;
  END_VAR
  FOR i:=_FIRST_AXIS#FIRST_AXIS TO _FIRST_AXIS#FIRST_AXIS+_MAXIS#MAXAXIS-1 DO
    pm[i].MA_LIMITE_ATTIVO:=1;
    IF i<>PrimoAsseNoGestione AND i<>SecondoAsseNoGestione AND
       i<>TerzoAsseNoGestione AND i<>QuartoAsseNoGestione AND
       i<>QuintoAsseNoGestione AND i<>SestoAsseNoGestione THEN
			(*{
			#ifdef ELECTXL
			}*)
				IF i=Q1 OR i=V1 THEN
					//Per ELECT-XL occorre gestire i limiti degli assi Q1 e V1 quando è abilitato da VGP
					//l^accessorio
					Eseguire:=Set_Limiti_Q1V1()=FALSE ;
				END_IF;
			(*{
			#endif //Fine ELECTXL
			}*)
			IF Eseguire=TRUE THEN
				//Se non sono in monitoring attivo i limiti software 1 agli assi, considerando la posizione
				//attuale del^asse
				ImpostaLimiteSW(Asse:=i, ValoreMinus:=pm[i].Ma_Pos_Limit_Minus_Attivo-EXTRALIMIT);
				ImpostaLimiteSW(Asse:=i, ValorePlus:=pm[i].Ma_Pos_Limit_Plus_Attivo+EXTRALIMIT);
			END_IF;
    END_IF;
  END_FOR;
END_FUNCTION

/**********************************************************************************************************************
 *           WITH ACCESSORY MO00003632 (INCREASE AXIS TRAVEL Q1 FOR MEDIUM RADIUS UP TO 610MM, THE TRAVELS            *
 *                                   OF Q1 AND V1 ACCORDING TO THE FOLLOWING RULES:                                   *
 *      - MAXIMUM LIMIT INCREASE OF Q1, INDICATED BY VGP VIA THE VARIABLE CFG.LIMQ1CAUSATODAV1, IF THE POSITION       *
 *              OF V1 IS HIGHER THAN THE POSITION INDICATED BY VGP IN THE VARIABLE CFG.LIMV1CAUSATODAQ1               *
 *      - RECORDING OF THE STANDARD POSITIVE LIMIT OF Q1, INDICATED IN PARAMETER M36110, WHEN THE POSITION OF V1      *
 *                   IS LOWER THAN THE VALUE INDICATED BY VGP IN THE VARIABLE CFG.LIMV1CAUSATODAQ1                    *
 * - REDUCTION OF THE NEGATIVE LIMIT OF V1 TO THE VALUE INDICATED BY VGP IN THE VARIABLE CFG.LIMV1CAUSATODAQ1, IF THE *
 *           POSITION OF Q1 IS HIGHER THAN THE STANDARD POSITIVE LIMIT INDICATED IN THE PARAMETER IN M36110           *
 *   - REDETERMINATION OF THE STANDARD NEGATIVE LIMIT OF V1, INDICATED IN PARAMETER M36110, WHEN THE POSITION OF Q1   *
 *                         IS LOWER THAN THE POSITIVE LIMIT OF Q1 GIVEN IN PARAMETER M36110.                          *
 **********************************************************************************************************************/

 (*{
#ifdef ELECTXL
}*)
	FUNCTION Set_Limiti_Q1V1:BOOL

    VAR_EXTERNAL
    cfg                             :_TYPE.Config_Struct;
    pm                              : ARRAY[_FIRST_AXIS#FIRST_AXIS.._FIRST_AXIS#FIRST_AXIS+_CONST_VAR_DEF._MAXIS#MAXAXIS-1] OF AxisParameters;
    Axes                            :ARRAY[_FIRST_AXIS#FIRST_AXIS.._FIRST_AXIS#FIRST_AXIS+_CONST_VAR_DEF._MAXIS#MAXAXIS-1] OF ax;/// ax as structure is defined in _TYPE
  END_VAR

    VAR_EXTERNAL CONSTANT
      EXTRALIMIT         	                :REAL; // extralimite per limiti fisici
      MY_BIG_VALUE_REAL                   :REAL;
      V1 : INT;
      Q1 : INT;
    END_VAR

    VAR
      PosAx : REF_TO TO_SynchronousAxis;
    END_VAR

		IF cfg.LimQ1CausatoDaV1<MY_BIG_VALUE_REAL-1 AND cfg.LimQ1CausatoDaV1<>-1 AND
			 cfg.LimV1CausatoDaQ1<MY_BIG_VALUE_REAL-1 AND cfg.LimV1CausatoDaQ1<>-1 THEN
			//Gestione limite V1 in funzione della posizione di Q1
      PosAx := AsSynchronousAxisRef(Axes[Q1].PosAx);
			IF PosAx^.ActualPosition>pm[Q1].Ma_Pos_Limit_Plus THEN
				ImpostaLimiteSw(Asse:=V1, ValoreMinus:=cfg.LimV1CausatoDaQ1-EXTRALIMIT);
			ELSE
				ImpostaLimiteSw(Asse:=V1, ValoreMinus:=pm[V1].Ma_Pos_Limit_Minus-EXTRALIMIT);
			END_IF;
			//Gestione limite Q1 in funzione della posizione di V1
      PosAx := AsSynchronousAxisRef(Axes[V1].PosAx);
			IF PosAx^.ActualPosition>cfg.LimV1CausatoDaQ1 THEN
				ImpostaLimiteSw(Asse:=Q1, ValorePlus:=cfg.LimQ1CausatoDaV1+EXTRALIMIT);
			ELSE
				ImpostaLimiteSw(Asse:=Q1, ValorePlus:=pm[Q1].Ma_Pos_Limit_Plus+EXTRALIMIT);
			END_IF;
			Set_Limiti_Q1V1:=TRUE;
		ELSE
			Set_Limiti_Q1V1:=FALSE;
		END_IF;
	END_FUNCTION
(*{
#endif //FINE ELECTXL
}*)

/****************************************************
 * TRUE IF THE INDICATED AXLE IS READY FOR MOVEMENT *
 ****************************************************/

FUNCTION TestAssePronto:BOOL

  VAR_EXTERNAL
    Axes                            :ARRAY[_FIRST_AXIS#FIRST_AXIS.._FIRST_AXIS#FIRST_AXIS+_CONST_VAR_DEF._MAXIS#MAXAXIS-1] OF ax;/// ax as structure is defined in _TYPE
  END_VAR

  VAR_INPUT
    Asse  :INT;
  END_VAR
  ;
  // IF  CheckIfTOactive(Axis:=Asse)=TRUE THEN %%%%%
  //   IF Axes[Asse].PosAx.actormonitoring.drivestate=ACTIVE AND
  //      Axes[Asse].PosAx.actormonitoring.power=ACTIVE THEN
  //     TestAssePronto:=TRUE;
  //   ELSE
  //     TestAssePronto:=FALSE;
  //   END_IF;
  // END_IF;
END_FUNCTION

/*******************************************************************
 * REACTIVATION OF OUTPUTS WHICH MUST BE RESET WITH CYCLE STOP AND *
 *     SUBSEQUENTLY RESET WITH THE VALUE MEMORISED WITH START      *
 *******************************************************************/

FUNCTION OffStopCicloDispositivi

  VAR_EXTERNAL
    i_sys_stopcond      : INT; // 0=NO STOP, 1=STOP ATTIVO
  END_VAR

  VAR_EXTERNAL CONSTANT
    MAXDIGITALOUTPUT                    :INT;
    OAddress                        : ARRAY [0..MAXDIGITALOUTPUT] OF Digital_Output;
  END_VAR
  VAR
    i    :DINT;
  END_VAR;
  FOR i:=0 TO MAXDIGITALOUTPUT DO
    IF oaddress[i].AbilGestStopCiclo=TRUE AND
       i_sys_stopcond=0 AND
       oaddress[i].StatoPreStopCiclo=TRUE THEN
      WriteDigitalOutput(NumOutput:=i, Value:=oaddress[i].statoprestopciclo);
      oaddress[i].statoprestopciclo:=FALSE;
    END_IF;
  END_FOR;
END_FUNCTION

FUNCTION ResetAllOutStopPoint

  VAR_EXTERNAL CONSTANT
    PRIMO_STOP_POINT_SET_OUT              	:INT;
    MAX_INP_OUT_STOP_POINT                  :INT;
    PRIMO_STOP_POINT_RESET_OUT            	:INT; //252
    ULTIMO_STOP_POINT_SET_OUT             	:INT;//251
    ULTIMO_STOP_POINT_RESET_OUT           	:INT;//275
  END_VAR

  VAR
    i :INT;
  END_VAR
  FOR i:=PRIMO_STOP_POINT_RESET_OUT TO ULTIMO_STOP_POINT_RESET_OUT DO
    OutStopPoint(Codice:=i, Stato:=FALSE);
  END_FOR;
END_FUNCTION

/*************************************
 * SETTING COMMAND OUTPUTS FROM STOP *
 *************************************/
FUNCTION OutStopPoint

  VAR_EXTERNAL CONSTANT
    PRIMO_STOP_POINT_SET_OUT              	:INT;
    MAX_INP_OUT_STOP_POINT                  :INT;
    PRIMO_STOP_POINT_RESET_OUT            	:INT; //252
    ULTIMO_STOP_POINT_SET_OUT             	:INT;//251
    ULTIMO_STOP_POINT_RESET_OUT           	:INT;//275
    ADDRES_OUT_STOPP: ARRAY[PRIMO_STOP_POINT_SET_OUT..ULTIMO_STOP_POINT_SET_OUT] OF INT;
  END_VAR

  VAR_INPUT
    Codice  :LREAL;
    Stato   :BOOL;
  END_VAR
  VAR
    i       :INT;
    dret    :DINT;
  END_VAR
  IF Stato=TRUE THEN
    FOR i:=PRIMO_STOP_POINT_SET_OUT TO ULTIMO_STOP_POINT_SET_OUT DO
      IF Codice=i THEN
        WriteDigitalOutput(NumOutput:=ADDRES_OUT_STOPP[TO_INT(Codice)], Value:=Stato);
      END_IF;
    END_FOR;
  ELSE
    FOR i:=PRIMO_STOP_POINT_RESET_OUT TO ULTIMO_STOP_POINT_RESET_OUT DO
      IF Codice=i THEN
        WriteDigitalOutput(NumOutput:=ADDRES_OUT_STOPP[TO_INT(Codice-MAX_INP_OUT_STOP_POINT)], Value:=Stato);
      END_IF;
    END_FOR;
  END_IF;
END_FUNCTION

FUNCTION Set_Disp

  VAR_EXTERNAL
    Disp                            :ARRAY[(FIRST_DEVICE)..(FIRST_DEVICE+_MAXDEVICES#MAXDEVICES-1)] OF Device;
    OAddress                        : ARRAY [0..MAXDIGITALOUTPUT] OF Digital_Output;
    MinutiRisparmioEnergetico       :INT;
  END_VAR

  VAR_EXTERNAL CONSTANT
    FIRST_DEVICE                          :INT;
    MAXDIGITALOUTPUT                      :INT;
    DISP_IN_TT                            :SINT;		//01 - TEMPO LAVORO - TEMPO RIPOSO   xxxxxxx0001
    DISP_IN_TM                            :SINT;		//03 - TEMPO LAVORO - MICRO RIPOSO   xxxxxxx0011
    DISP_IN_MT                            :SINT;		//05 - MICRO LAVORO - TEMPO RIPOSO   xxxxxxx0101
    DISP_IN_MM                            :SINT;		//07 - MICRO LAVORO - MICRO RIPOSO   xxxxxxx0111
    DISP_IN_AI	                          :SINT;		//09 - INGRESSO ANALOGICO      xxxxxxx1001
    DISP_IN_V                             :SINT;	//16 - INGRESSO VIRTUALE       xxxxxx10000 COMANDATO DALLA LOGICA INTERNA (es: un altro task)

    DISP_OUT_DO                           :SINT;		//1 - USCITA DIGITALE         xxxxxxxxx01
    DISP_OUT_AO                           :SINT; 	//3 - USCITA ANALOGICA        xxxxxxxxx11

  END_VAR

  VAR_INPUT
    Ndisp            :INT;
    Stato            :INT;
    TimerRisparmio  :BOOL;
  END_VAR
  VAR
    Valore          :REAL;
    dret            :DINT;
  END_VAR
  Disp[Ndisp].StatoRichiesto:=Stato;
  IF Disp[NDisp].Enable=FALSE THEN ;
    oaddress[Ndisp].stato:=FALSE;
    // GOTO End;
  END_IF;
  IF TimerRisparmio=TRUE THEN
    StartTimerRisparmioEnergetico(Tempo:=MinutiRisparmioEnergetico);
  END_IF;
  CASE Disp[Ndisp].TipoOut OF
    DISP_OUT_DO:
      IF Disp[Ndisp].spegnimentouscita=TRUE THEN
        IF Disp[Ndisp].Stato=Disp[Ndisp].StatoRichiesto THEN ;
          // GOTO End;
        END_IF;
      END_IF;
      IF Stato=DEVICES_STATUS#LAVORO THEN
        WriteDigitalOutput(NumOutput:=DISP[Ndisp].Out_Riposo, Value:=FALSE);
        WriteDigitalOutput(NumOutput:=DISP[Ndisp].Out_Riposo_2, Value:=FALSE);
        IF DISP[Ndisp].Ritardo_Uscite>0 THEN
          WriteDigitalOutput(NumOutput:=DISP[Ndisp].Out_Lavoro, Value:=TRUE);
          //dret:=_waitTime(timeValue:=REAL_TO_TIME(DISP[Ndisp].Ritardo_Uscite*1000));
          WriteDigitalOutput(NumOutput:=DISP[Ndisp].Out_Lavoro_2, Value:=TRUE);
        ELSE
          WriteDigitalOutput(NumOutput:=DISP[Ndisp].Out_Lavoro_2, Value:=TRUE);
          //dret:=_waitTime(timeValue:=REAL_TO_TIME(ABS(DISP[Ndisp].Ritardo_Uscite*1000)));
          WriteDigitalOutput(NumOutput:=DISP[Ndisp].Out_Lavoro, Value:=TRUE);
        END_IF;
      ELSE
        IF Stato=DEVICES_STATUS#RIPOSO THEN
          WriteDigitalOutput(NumOutput:=DISP[Ndisp].Out_Lavoro, Value:=FALSE);
          WriteDigitalOutput(NumOutput:=DISP[Ndisp].Out_Lavoro_2, Value:=FALSE);
          WriteDigitalOutput(NumOutput:=DISP[Ndisp].Out_Riposo, Value:=TRUE);
          WriteDigitalOutput(NumOutput:=DISP[Ndisp].Out_Riposo_2, Value:=TRUE);
        END_IF;
      END_IF;
    DISP_OUT_AO:;
      //Uscita analogica
  END_CASE;
  //Muove solo se non si trova già sullo stato finale
  IF Stato<>DISP[Ndisp].Stato THEN
    //Doppia uscita digitale
    CASE DISP[Ndisp].TipoIn OF
      DISP_IN_TT:
        //Tempo lavoro, Tempo riposo
        IF Stato=DEVICES_STATUS#LAVORO THEN
          IF Disp[NDisp].Stato<>DEVICES_STATUS#VERSO_LAVORO OR NOT DISP[NDisp].In_Movimento THEN
            DISP[NDisp].Timer:=((DISP[Ndisp].limite_Lavoro-DISP[Ndisp].Position)/DISP[Ndisp].Vel_Lavoro*1000);
          END_IF;
          Disp[NDisp].Stato:=DEVICES_STATUS#VERSO_LAVORO;
          DISP[NDisp].In_Movimento:=TRUE;
        ELSE
          IF Stato=DEVICES_STATUS#RIPOSO THEN
            IF Disp[NDisp].Stato<>DEVICES_STATUS#VERSO_RIPOSO OR NOT DISP[NDisp].In_Movimento THEN
              DISP[NDisp].Timer:=(DISP[Ndisp].Position-DISP[Ndisp].Limite_Riposo)/DISP[Ndisp].Vel_Riposo*1000;
            END_IF;
            Disp[NDisp].Stato:=DEVICES_STATUS#VERSO_RIPOSO;
            DISP[NDisp].In_Movimento:=TRUE;
          END_IF;
        END_IF;
      DISP_IN_TM:  // 3  - TEMPO LAVORO - MICRO RIPOSO   xxxxxxx0011
        IF Stato=DEVICES_STATUS#LAVORO THEN
          IF Disp[NDisp].Stato<>DEVICES_STATUS#VERSO_LAVORO OR NOT DISP[NDisp].In_Movimento THEN
            DISP[NDisp].Timer:=((DISP[Ndisp].Limite_Lavoro-DISP[Ndisp].Position)/DISP[Ndisp].Vel_Lavoro*1000);
          END_IF;
          Disp[NDisp].Stato:=DEVICES_STATUS#VERSO_LAVORO;
          DISP[NDisp].In_Movimento:=TRUE;
        ELSE
          IF Stato=DEVICES_STATUS#RIPOSO THEN
            IF Disp[NDisp].Stato<>DEVICES_STATUS#VERSO_RIPOSO OR NOT DISP[NDisp].In_Movimento THEN
              DISP[NDisp].Timer:=((DISP[Ndisp].Position-DISP[Ndisp].Limite_Riposo)/DISP[Ndisp].Vel_Lavoro*1000);
            END_IF;
            DISP[NDisp].In_Movimento:=TRUE;
            Disp[NDisp].Stato:=DEVICES_STATUS#VERSO_RIPOSO;
          END_IF;
        END_IF;
      DISP_IN_MT:  // 5  - MICRO LAVORO - TEMPO RIPOSO   xxxxxxx0101
        IF Stato=DEVICES_STATUS#LAVORO THEN
          IF Disp[NDisp].Stato<>DEVICES_STATUS#VERSO_LAVORO OR NOT DISP[NDisp].In_Movimento THEN
            DISP[NDisp].Timer:=((DISP[Ndisp].Limite_Lavoro-DISP[Ndisp].Position)/DISP[Ndisp].Vel_Lavoro*1000);
          END_IF;
          DISP[NDisp].In_Movimento:=TRUE;
          Disp[NDisp].Stato:=DEVICES_STATUS#VERSO_LAVORO;
         ELSE
          IF Stato=DEVICES_STATUS#RIPOSO THEN
            IF Disp[NDisp].Stato<>DEVICES_STATUS#VERSO_RIPOSO OR NOT DISP[NDisp].In_Movimento THEN
              DISP[NDisp].Timer:=(DISP[Ndisp].Position-DISP[Ndisp].Limite_Riposo)/DISP[Ndisp].Vel_Lavoro*1000;
            END_IF;
              DISP[NDisp].In_Movimento:=TRUE;
              Disp[NDisp].Stato:=DEVICES_STATUS#VERSO_RIPOSO;
            END_IF;
        END_IF;
      DISP_IN_MM:  // 7  - MICRO LAVORO - MICRO RIPOSO   xxxxxxx0111
        DISP[NDisp].In_Movimento:=TRUE;
        IF Stato=DEVICES_STATUS#LAVORO THEN
          Disp[NDisp].Stato:=DEVICES_STATUS#VERSO_LAVORO;
          DISP[NDisp].Timer:=((DISP[Ndisp].Limite_Lavoro-DISP[Ndisp].Position)/DISP[Ndisp].Vel_Lavoro*1000);
        ELSE
          IF Stato=DEVICES_STATUS#RIPOSO THEN
            Disp[NDisp].Stato:=DEVICES_STATUS#VERSO_RIPOSO;
            DISP[NDisp].Timer:=(DISP[Ndisp].Position-DISP[Ndisp].Limite_Riposo)/DISP[Ndisp].Vel_Lavoro*1000;
          END_IF;
        END_IF;
       DISP_IN_AI:;  // 9  - INGRESSO ANALOGICO      xxxxxxx1001
       DISP_IN_V:;  // 16  - INGRESSO VIRTUALE
       DISP[NDisp].In_Movimento:=TRUE;
    END_CASE;
    //Incremento del timer del valore del filtro
    DISP[NDisp].Timer:=DISP[NDisp].Timer+(Disp[Ndisp].timerfiltro*1000);
  ELSE
    DISP[NDisp].In_Movimento:=FALSE;
  END_IF;
  // {
  // #ifdef ELECTL_ALL %%%%
  // }
    // Set_Disp_ElectL(Ndisp,Stato);
  // {
  // #endif  //Fine ELECTL_ALL
  // }
  // {
  // #ifdef ELECTXL %%%%
  // }
  //   Set_Disp_ElectXL(Ndisp,Stato);
  // {
  // #endif  //Fine ELECTXL
  // }
  //End:;
END_FUNCTION

FUNCTION SetDispComplesso

  VAR_EXTERNAL
    MinutiRisparmioEnergetico               :INT;
    cfg                                     :_TYPE.Config_Struct;
    Disp                                    :ARRAY[(FIRST_DEVICE)..(FIRST_DEVICE+_MAXDEVICES#MAXDEVICES-1)] OF Device;
  END_VAR

  VAR_EXTERNAL CONSTANT
    CILSOTTOTESTA                                 :INT;
    SUPPORT_TIRANT                                :INT;
    FIRST_DEVICE                                  :INT;
    OUT_CHIUSURA_CILINDRO_SOTTOTESTA              :INT;
    OUT_APERTURA_CILINDRO_SOTTOTESTA              :INT;
    OUT_APERTURA_INTERMEDIA_CILINDRO_SOTTOTESTA   :INT;
  END_VAR

  VAR_INPUT
    Ndisp           :INT;
    Value           :REAL;
    Attesa          :BOOL;
    TimerRisparmio  :BOOL;

  END_VAR

  VAR
    dret            :DINT;
    ProgrammaAttivo :DINT;
    Stato           :INT;
		AppoValue				:REAL;
  END_VAR

  IF TimerRisparmio=TRUE THEN
    StartTimerRisparmioEnergetico(Tempo:=MinutiRisparmioEnergetico);
  END_IF;
  // {
  // #ifdef ORBITALE %%%%
  // }
  //   {
  //   #ifdef DH4010
  //   }
	// 		CASE Ndisp OF
	// 			BLOCCAGGIO_2D:
	// 				IF Disp[NDisp].Enable=FALSE THEN
	// 					Disp[Ndisp].in_movimento:=FALSE;
	// 					oaddress[OUT_CHIUSURA_RESISTENZA_1].stato:=FALSE;
	// 					oaddress[OUT_CHIUSURA_RESISTENZA_2].stato:=FALSE;
	// 					oaddress[OUT_CHIUSURA_RESISTENZA_3].stato:=FALSE;
	// 					oaddress[OUT_CHIUSURA_RESISTENZA_4].stato:=FALSE;
	// 					oaddress[OUT_APERTURA_RESISTENZA_1].stato:=FALSE;
	// 					oaddress[OUT_APERTURA_RESISTENZA_2].stato:=FALSE;
	// 					oaddress[OUT_APERTURA_RESISTENZA_3].stato:=FALSE;
	// 					oaddress[OUT_APERTURA_RESISTENZA_4].stato:=FALSE;
	// 				ELSE
	// 					IF Disp[Ndisp].StatoRichiesto=Disp[Ndisp].stato THEN
	// 						Disp[Ndisp].in_movimento:=FALSE;
	// 					ELSE
	// 						Disp[Ndisp].in_movimento:=TRUE;
	// 					END_IF;
	// 					CASE Value OF
	// 						RIPOSO:
	// 							//Apertura tutte insieme
	// 							Set_Disp(Ndisp:=BLOCCAGGIO_RESISTENZA_1, Stato:=RIPOSO, TimerRisparmio:=TRUE);
	// 							Set_Disp(Ndisp:=BLOCCAGGIO_RESISTENZA_2, Stato:=RIPOSO, TimerRisparmio:=TRUE);
	// 							Set_Disp(Ndisp:=BLOCCAGGIO_RESISTENZA_3, Stato:=RIPOSO, TimerRisparmio:=TRUE);
	// 							Set_Disp(Ndisp:=BLOCCAGGIO_RESISTENZA_4, Stato:=RIPOSO, TimerRisparmio:=TRUE);
	// 						LAVORO:
	// 							//Chiusura delle sole posizioni abilitate
	// 							IF Centratore_cfg.ResistenzeProg[0]=TRUE THEN
	// 								Set_Disp(Ndisp:=BLOCCAGGIO_RESISTENZA_1, Stato:=LAVORO, TimerRisparmio:=TRUE);
	// 							END_IF;
	// 							IF Centratore_cfg.ResistenzeProg[1]=TRUE THEN
	// 								Set_Disp(Ndisp:=BLOCCAGGIO_RESISTENZA_2, Stato:=LAVORO, TimerRisparmio:=TRUE);
	// 							END_IF;
	// 							IF Centratore_cfg.ResistenzeProg[2]=TRUE THEN
	// 								Set_Disp(Ndisp:=BLOCCAGGIO_RESISTENZA_3, Stato:=LAVORO, TimerRisparmio:=TRUE);
	// 							END_IF;
	// 							IF Centratore_cfg.ResistenzeProg[3]=TRUE THEN
	// 								Set_Disp(Ndisp:=BLOCCAGGIO_RESISTENZA_4, Stato:=LAVORO, TimerRisparmio:=TRUE);
	// 							END_IF;
	// 					END_CASE;
	// 				END_IF;
	// 			PINZA_SX:
	// 				IF Disp[NDisp].Enable=FALSE THEN ;
	// 					oaddress[OUT_PINZA_PRECHIUSA1_TESTA_SX].stato:=FALSE;
	// 					oaddress[OUT_PINZA_APERTA_TESTA_SX].stato:=FALSE;
	// 				ELSE
	// 					IF Disp[Ndisp].statorichiesto<>Disp[Ndisp].stato THEN
	// 						IF ((Disp[Ndisp].stato=LAVORO AND mcpi_minus=TRUE) OR
	// 								(Disp[Ndisp].stato=RIPOSO AND mcpi_plus=TRUE) OR
	// 								(Disp[Ndisp].stato<>LAVORO AND Disp[Ndisp].stato<>RIPOSO) OR
	// 								(i_sys_activedevice=C_TAGLIO_SX) OR (i_sys_activedevice=CMD_CURVA_MANUALE) OR (i_sys_activedevice=CMD_SNERVAMENTO) OR (i_sys_activedevice=CMD_FINE_SNERVAMENTO)) OR
	// 								i_sys_OPMODE<>JOGMODE THEN
	// 							//Se è attivo il JOG la gestione dei tasti + o - deve essere condizionata allo stato
	// 							//di partenza del dispositivo
	// 							Disp[Ndisp].in_movimento:=TRUE;
	// 							//In caso di posizione indefinita si esegue comunque l^apertura
	// 							IF Disp[Ndisp].Position=INDEFINITO AND i_sys_opmode=JOGMODE AND i_sys_activedevice=Ndisp THEN
	// 								AppoValue:=RIPOSO;
	// 							ELSE
	// 								AppoValue:=Value;
	// 							END_IF;
	// 							CASE AppoValue OF
	// 								RIPOSO:
	// 									//Apertura pinza
	// 									WriteDigitalOutput(NumOutput:=OUT_PINZA_PRECHIUSA1_TESTA_SX, Value:=FALSE);
	// 									WriteDigitalOutput(NumOutput:=OUT_PINZA_APERTA_TESTA_SX, Value:=TRUE);
	// 									Set_Disp(Ndisp:=PINZA_SX_PRECHIUSURA, Stato:=RIPOSO, TimerRisparmio:=TRUE);
	// 								INTERMEDIO_PINZA:
	// 									//Prechiusura pinza
	// 									WriteDigitalOutput(NumOutput:=OUT_PINZA_PRECHIUSA1_TESTA_SX, Value:=TRUE);
	// 									WriteDigitalOutput(NumOutput:=OUT_PINZA_APERTA_TESTA_SX, Value:=FALSE);
	// 									Set_Disp(Ndisp:=PINZA_SX_PRECHIUSURA, Stato:=RIPOSO, TimerRisparmio:=TRUE);
	// 								LAVORO:
	// 									//Chiusura pinza
	// 									WriteDigitalOutput(NumOutput:=OUT_PINZA_PRECHIUSA1_TESTA_SX, Value:=TRUE);
	// 									WriteDigitalOutput(NumOutput:=OUT_PINZA_APERTA_TESTA_SX, Value:=FALSE);
	// 									Set_Disp(Ndisp:=PINZA_SX_PRECHIUSURA, Stato:=LAVORO, TimerRisparmio:=TRUE);
	// 							END_CASE;
	// 						END_IF;
	// 					END_IF;
	// 				END_IF;
	// 			PINZA_DX:
	// 				IF Disp[NDisp].Enable=FALSE THEN ;
	// 					oaddress[OUT_PINZA_PRECHIUSA1_TESTA_DX].stato:=FALSE;
	// 					oaddress[OUT_PINZA_APERTA_TESTA_DX].stato:=FALSE;
	// 				ELSE
	// 					IF Disp[Ndisp].statorichiesto<>Disp[Ndisp].stato THEN
	// 						IF ((Disp[Ndisp].stato=LAVORO AND mcpi_minus=TRUE) OR
	// 								(Disp[Ndisp].stato=RIPOSO AND mcpi_plus=TRUE) OR
	// 								(Disp[Ndisp].stato<>LAVORO AND Disp[Ndisp].stato<>RIPOSO) OR
	// 								(i_sys_activedevice=C_TAGLIO_DX) OR (i_sys_activedevice=CMD_CURVA_MANUALE) OR (i_sys_activedevice=CMD_SNERVAMENTO) OR (i_sys_activedevice=CMD_FINE_SNERVAMENTO)) OR
	// 							 i_sys_OPMODE<>JOGMODE THEN
	// 							//Se è attivo il JOG la gestione dei tasti + o - deve essere condizionata allo stato
	// 							//di partenza del dispositivo
	// 							Disp[Ndisp].in_movimento:=TRUE;
	// 							//In caso di posizione indefinita si esegue comunque l^apertura
	// 							IF Disp[Ndisp].Position=INDEFINITO AND i_sys_opmode=JOGMODE AND i_sys_activedevice=Ndisp THEN
	// 								AppoValue:=RIPOSO;
	// 							ELSE
	// 								AppoValue:=Value;
	// 							END_IF;
	// 							CASE AppoValue OF
	// 								RIPOSO:
	// 									//Apertura pinza
	// 									WriteDigitalOutput(NumOutput:=OUT_PINZA_PRECHIUSA1_TESTA_DX, Value:=FALSE);
	// 									WriteDigitalOutput(NumOutput:=OUT_PINZA_APERTA_TESTA_DX, Value:=TRUE);
	// 									Set_Disp(Ndisp:=PINZA_DX_PRECHIUSURA, Stato:=RIPOSO, TimerRisparmio:=TRUE);
	// 								INTERMEDIO_PINZA:
	// 									//Prechiusura pinza
	// 									WriteDigitalOutput(NumOutput:=OUT_PINZA_PRECHIUSA1_TESTA_DX, Value:=TRUE);
	// 									WriteDigitalOutput(NumOutput:=OUT_PINZA_APERTA_TESTA_DX, Value:=FALSE);
	// 									Set_Disp(Ndisp:=PINZA_DX_PRECHIUSURA, Stato:=RIPOSO, TimerRisparmio:=TRUE);
	// 								LAVORO:
	// 									//Chiusura pinza
	// 									WriteDigitalOutput(NumOutput:=OUT_PINZA_PRECHIUSA1_TESTA_DX, Value:=TRUE);
	// 									WriteDigitalOutput(NumOutput:=OUT_PINZA_APERTA_TESTA_DX, Value:=FALSE);
	// 									Set_Disp(Ndisp:=PINZA_DX_PRECHIUSURA, Stato:=LAVORO, TimerRisparmio:=TRUE);
	// 							END_CASE;
	// 						END_IF;
	// 					END_IF;
	// 				END_IF;
	// 			ELSE
  //       ;
  //     END_CASE;
  //   {
  //   #endif  //Fine DH4010
  //   }
  //   {
  //   #ifdef EFLEX
  //   }
  //     CASE Ndisp OF
  //       TESTINA_1, TESTINA_2:
  //         IF Disp[Ndisp].statorichiesto<>Disp[Ndisp].stato THEN
  //           Disp[Ndisp].in_movimento:=TRUE;
  //           CASE Value OF
  //             RIPOSO:
  //               //Sollevamento testina
  //               WriteDigitalOutput(NumOutput:=Disp[Ndisp].Out_Riposo, Value:=TRUE);
  //               WriteDigitalOutput(NumOutput:=Disp[Ndisp].Out_Lavoro, Value:=FALSE);
  //             INTERMEDIO:
  //               IF Disp[Ndisp].position=LAVORO THEN
  //                 //Si parte da testina bassa, si solleva la testina
  //                 WriteDigitalOutput(NumOutput:=Disp[Ndisp].Out_Riposo, Value:=TRUE);
  //                 WriteDigitalOutput(NumOutput:=Disp[Ndisp].Out_Lavoro, Value:=FALSE);
  //               ELSE
  //                 IF Disp[Ndisp].position=RIPOSO THEN
  //                   //Si parte da testina alta, si abbassa la testina
  //                   WriteDigitalOutput(NumOutput:=Disp[Ndisp].Out_Lavoro, Value:=TRUE);
  //                   WriteDigitalOutput(NumOutput:=Disp[Ndisp].Out_Riposo, Value:=FALSE);
  //                 END_IF;
  //               END_IF;
  //             LAVORO:
  //               //Abbassamento testina
  //               WriteDigitalOutput(NumOutput:=Disp[Ndisp].Out_Lavoro, Value:=TRUE);
  //               WriteDigitalOutput(NumOutput:=Disp[Ndisp].Out_Riposo, Value:=FALSE);
  //           END_CASE;
  //         END_IF;
  //     ELSE
  //       ;
  //     END_CASE;
  //   {
  //   #endif  //Fine EFLEX
  //   }
  //   {
  //   #ifdef RUNNER
  //   }
  //     CASE Ndisp OF
  //       RULLATORE:
  //         IF Disp[Ndisp].StatoRichiesto<>Disp[Ndisp].Stato OR Disp[Ndisp].StatoRichiesto<>Disp[Ndisp].Position THEN
  //           Disp[Ndisp].in_movimento:=TRUE;
  //           CASE Value OF
  //             LAVORO:
  //               //Rotazione veloce senso orario
  //               WriteDigitalOutput(NumOutput:=OUT_4RROT_MOTORE_INVERSIONE_ROTAZIONE, Value:=FALSE);
  //               WriteDigitalOutput(NumOutput:=OUT_4RROT_MOTORE_VEL_MIN, Value:=FALSE);
  //               WriteDigitalOutput(NumOutput:=OUT_4RROT_MOTORE_VEL_MAX, Value:=TRUE);
  //             INTERMEDIO:
  //               //Rotazione lenta senso orario
  //               WriteDigitalOutput(NumOutput:=OUT_4RROT_MOTORE_INVERSIONE_ROTAZIONE, Value:=FALSE);
  //               WriteDigitalOutput(NumOutput:=OUT_4RROT_MOTORE_VEL_MAX, Value:=FALSE);
  //               WriteDigitalOutput(NumOutput:=OUT_4RROT_MOTORE_VEL_MIN, Value:=TRUE);
  //           ELSE
  //             IF Value=-INTERMEDIO THEN
  //               //Rotazione lenta senso antiorario
  //               WriteDigitalOutput(NumOutput:=OUT_4RROT_MOTORE_VEL_MIN, Value:=FALSE);
  //               WriteDigitalOutput(NumOutput:=OUT_4RROT_MOTORE_VEL_MAX, Value:=FALSE);
  //               WriteDigitalOutput(NumOutput:=OUT_4RROT_MOTORE_INVERSIONE_ROTAZIONE, Value:=TRUE);
  //             ELSE
  //               //Arresto rullatore
  //               WriteDigitalOutput(NumOutput:=OUT_4RROT_MOTORE_VEL_MIN, Value:=FALSE);
  //               WriteDigitalOutput(NumOutput:=OUT_4RROT_MOTORE_VEL_MAX, Value:=FALSE);
  //               WriteDigitalOutput(NumOutput:=OUT_4RROT_MOTORE_INVERSIONE_ROTAZIONE, Value:=FALSE);
  //             END_IF;
  //           END_CASE;
  //         END_IF;
  //       {
  //       #ifdef ASPO_RUNNER
  //       }
	// 				ASPO:
	// 					IF IAddress[INP_INVERTER_ASPO_ON].Port=-1 THEN
	// 						//Gestione aspo senza inverter
	// 						IF i_sys_OpMode=AUTOMODE THEN
	// 							ProgrammaAttivo:=I_SYS_Current_Prog;
	// 						ELSE
	// 							ProgrammaAttivo:=PROGRAMMA_JOG;
	// 						END_IF;
	// 						IF cfg.ASPO_NuovoModo=TRUE THEN
	// 							IF programmi[ProgrammaAttivo].ModoAspo=ASPO_IN_FOLLE OR i_sys_SenzaTubo=TRUE THEN
	// 								//ASPO_IN_FOLLE
	// 								WriteDigitalOutput(NumOutput:=Disp[Ndisp].out_lavoro, Value:=FALSE);
	// 								WriteDigitalOutput(NumOutput:=Disp[Ndisp].out_riposo, Value:=FALSE);
	// 								WriteDigitalOutput(NumOutput:=OUT_4RASPO_PRESSIONE_FRIZIONE, Value:=FALSE);
	// 							ELSE
	// 								//ASPO_MOTORIZZATO o ASPO_IN_FOLLE_AVANZAMENTO
	// 								Disp[Ndisp].in_movimento:=TRUE;
	// 								CASE Value OF
	// 									LAVORO:
	// 										//Svolgimento aspo
	// 										IF programmi[ProgrammaAttivo].ModoAspo=ASPO_MOTORIZZATO THEN
	// 											//Svolgimento motorizzato si attiva la frizione
	// 											WriteDigitalOutput(NumOutput:=OUT_4RASPO_PRESSIONE_FRIZIONE, Value:=TRUE);
	// 										ELSE
	// 											//Svolgimento in folle si disattiva la frizione
	// 											WriteDigitalOutput(NumOutput:=OUT_4RASPO_PRESSIONE_FRIZIONE, Value:=FALSE);
	// 										END_IF;
	// 										IF readdigitalinput(NumInput:=Disp[Ndisp].in_lavoro, Verifica:=TRUE)=FALSE THEN
	// 											//Svolgimento tubo solo se braccio aspo non è aperto
	// 											WriteDigitalOutput(NumOutput:=Disp[Ndisp].out_riposo, Value:=FALSE);
	// 											IF programmi[ProgrammaAttivo].ModoAspo<>ASPO_IN_FOLLE_AVANZAMENTO OR
	// 												 OAddress[OUT_ASPO_VERTICALE_NO_ATTREZZAGGIO].port=-1 THEN
	// 												//Con aspo verticale non si deve attivare la valvola di svolgimento dell^aspo
	// 												//indicazione telefonica per cliente Bemasch di Alberto Pittioni 08/11/2017
	// 												WriteDigitalOutput(NumOutput:=Disp[Ndisp].out_lavoro, Value:=TRUE);
	// 											END_IF;
	// 										ELSE
	// 											//Con braccio aperto si ferma lo svolgimento dell^aspo e si aggancia comunque
	// 											//la frizione per eseguire la migliore frenatura possibile
	// 											WriteDigitalOutput(NumOutput:=OUT_4RASPO_PRESSIONE_FRIZIONE, Value:=TRUE);
	// 											WriteDigitalOutput(NumOutput:=Disp[Ndisp].out_lavoro, Value:=FALSE);
	// 										END_IF;
	// 									RIPOSO:
	// 										//Riavvolgimento aspo sempre motorizzato, sempre con frizione inserita
	// 										WriteDigitalOutput(NumOutput:=OUT_4RASPO_PRESSIONE_FRIZIONE, Value:=TRUE);
	// 										IF readdigitalinput(NumInput:=Disp[Ndisp].in_riposo, Verifica:=TRUE)=FALSE THEN
	// 											//Avvolgimento tubo solo se braccio aspo non è chiuso
	// 											WriteDigitalOutput(NumOutput:=Disp[Ndisp].out_lavoro, Value:=FALSE);
	// 											WriteDigitalOutput(NumOutput:=Disp[Ndisp].out_riposo, Value:=TRUE);
	// 										ELSE
	// 											//Con braccio chiuso si ferma l^avvolgimento dell^aspo
	// 											WriteDigitalOutput(NumOutput:=Disp[Ndisp].out_riposo, Value:=FALSE);
	// 										END_IF;
	// 									INTERMEDIO:
	// 										//Arresto aspo
	// 										IF cfg.ASPO_MantieneSvolgimento=FALSE OR
	// 											 i_sys_OPMODE<>AUTOMODE OR
	// 											 TestMasterLavoro()=FALSE OR
	// 											 OAddress[OUT_4RASPO_ASPO_SVOLGI_TUBO].stato=FALSE OR
	// 											 (cfg.ASPO_MantieneSvolgimento=TRUE AND
	// 												readdigitalinput(NumInput:=INP_ASPO_BRACCIO_APERTO, Verifica:=TRUE)=TRUE) THEN
	// 											//In automatico mantiene lo svolgimento dell^aspo fino all^attivazione
	// 											//del sensore di braccio aperto
	// 											WriteDigitalOutput(NumOutput:=OUT_4RASPO_PRESSIONE_FRIZIONE, Value:=TRUE);
	// 											WriteDigitalOutput(NumOutput:=Disp[Ndisp].out_lavoro, Value:=FALSE);
	// 											WriteDigitalOutput(NumOutput:=Disp[Ndisp].out_riposo, Value:=FALSE);
	// 										END_IF;
	// 								END_CASE;  //Case stati dell^Aspo
	// 							END_IF;
	// 						ELSE
	// 							//Vecchio modo
	// 							IF Disp[Ndisp].statorichiesto=Disp[Ndisp].stato THEN
	// 								IF Value=INTERMEDIO THEN
	// 									//Arresto aspo
	// 									WriteDigitalOutput(NumOutput:=Disp[Ndisp].out_lavoro, Value:=FALSE);
	// 									WriteDigitalOutput(NumOutput:=Disp[Ndisp].out_riposo, Value:=FALSE);
	// 								END_IF;
	// 							ELSE
	// 								//Aspo in movimento
	// 								Disp[Ndisp].in_movimento:=TRUE;
	// 								IF programmi[ProgrammaAttivo].ModoAspo=ASPO_IN_FOLLE THEN
	// 									//Richiesta rotazione in folle dell^aspo, si disabilita la frizione che trasmette il movimento
	// 									WriteDigitalOutput(NumOutput:=OUT_4RASPO_PRESSIONE_FRIZIONE, Value:=FALSE);
	// 								ELSE
	// 									//Richiesta rotazione standard dell^aspo, si abilita la frizione che trasmette il movimento
	// 									WriteDigitalOutput(NumOutput:=OUT_4RASPO_PRESSIONE_FRIZIONE, Value:=TRUE);
	// 								END_IF;
	// 								CASE Value OF
	// 									LAVORO:
	// 										IF readdigitalinput(NumInput:=Disp[Ndisp].in_lavoro, Verifica:=TRUE)=FALSE THEN
	// 											//Svolgimento tubo solo se braccio aspo non è aperto
	// 											IF i_sys_SenzaTubo=TRUE THEN
	// 												WriteDigitalOutput(NumOutput:=Disp[Ndisp].out_riposo, Value:=FALSE);
	// 												WriteDigitalOutput(NumOutput:=Disp[Ndisp].out_lavoro, Value:=FALSE);
	// 											ELSE
	// 												WriteDigitalOutput(NumOutput:=Disp[Ndisp].out_riposo, Value:=FALSE);
	// 												WriteDigitalOutput(NumOutput:=Disp[Ndisp].out_lavoro, Value:=TRUE);
	// 											END_IF;
	// 										END_IF;
	// 									RIPOSO:
	// 										IF readdigitalinput(NumInput:=Disp[Ndisp].in_riposo, Verifica:=TRUE)=FALSE THEN
	// 											//Avvolgimento tubo solo se braccio aspo non è chiuso
	// 											IF i_sys_SenzaTubo=TRUE THEN
	// 												WriteDigitalOutput(NumOutput:=Disp[Ndisp].out_lavoro, Value:=FALSE);
	// 												WriteDigitalOutput(NumOutput:=Disp[Ndisp].out_riposo, Value:=FALSE);
	// 											ELSE
	// 												WriteDigitalOutput(NumOutput:=Disp[Ndisp].out_lavoro, Value:=FALSE);
	// 												WriteDigitalOutput(NumOutput:=Disp[Ndisp].out_riposo, Value:=TRUE);
	// 											END_IF;
	// 										END_IF;
	// 									INTERMEDIO:
	// 										//Arresto aspo
	// 										WriteDigitalOutput(NumOutput:=Disp[Ndisp].out_lavoro, Value:=FALSE);
	// 										WriteDigitalOutput(NumOutput:=Disp[Ndisp].out_riposo, Value:=FALSE);
	// 								END_CASE;  //Case stati dell^Aspo
	// 							END_IF;
	// 						END_IF;
	// 					END_IF;
	// 				{
	// 				#endif	//Fine ASPO_RUNNER
	// 				}
  //       {
  //       #ifdef THREE_RUNNER
  //       }
  //         IPC_STRAPPO_SCARICO:
  //           IF Disp[Ndisp].statorichiesto<>Disp[Ndisp].stato THEN
  //             Disp[Ndisp].in_movimento:=TRUE;
  //           END_IF;
  //           //Per evitare che rimbalzi del sensore che rileva la posizione arretrata dello
  //           //strappo_scarico, si esegue comunque l^impostazione delle uscite
  //           CASE Value OF
  //             LAVORO:
  //               WriteDigitalOutput(NumOutput:=OUT_STRAPPO_SCARICO_AVANTI, Value:=TRUE);
  //               WriteDigitalOutput(NumOutput:=OUT_STRAPPO_SCARICO_INTERMEDIO, Value:=TRUE);
  //             RIPOSO:
  //               WriteDigitalOutput(NumOutput:=OUT_STRAPPO_SCARICO_INTERMEDIO, Value:=FALSE);
  //               WriteDigitalOutput(NumOutput:=OUT_STRAPPO_SCARICO_AVANTI, Value:=FALSE);
  //             INTERMEDIO:
  //               WriteDigitalOutput(NumOutput:=OUT_STRAPPO_SCARICO_AVANTI, Value:=FALSE);
  //               WriteDigitalOutput(NumOutput:=OUT_STRAPPO_SCARICO_INTERMEDIO, Value:=TRUE);
  //           END_CASE;
  //       {
  //       #endif  //Fine THREE_RUNNER
  //       }
  //       {
  //       #ifdef FOUR_RUNNER_PLAUNO
  //       }
  //         {
  //         #ifdef PLAUNO_PLAUNO_LIGHT
  //         }
  //           BLOCCAGGIO_TUBO:
  //             IF Disp[Ndisp].statorichiesto<>Disp[Ndisp].stato THEN
  //               Disp[Ndisp].in_movimento:=TRUE;
  //               Stato:=LREAL_TO_INT(Disp[Ndisp].statorichiesto);
  //               IF Stato=INTERMEDIO THEN
  //                 IF Assi[Q1].PosAx.positioningState.actualPosition>0.1 THEN
  //                   Set_Disp(Ndisp:=BLOCCAGGIO_TUBO_DX, Stato:=LAVORO, TimerRisparmio:=TRUE);
  //                   Set_Disp(Ndisp:=BLOCCAGGIO_TUBO_SX, Stato:=RIPOSO, TimerRisparmio:=TRUE);
  //                 ELSE
  //                   Set_Disp(Ndisp:=BLOCCAGGIO_TUBO_DX, Stato:=RIPOSO, TimerRisparmio:=TRUE);
  //                   Set_Disp(Ndisp:=BLOCCAGGIO_TUBO_SX, Stato:=LAVORO, TimerRisparmio:=TRUE);
  //                 END_IF;
  //               ELSE
  //                 Set_Disp(Ndisp:=BLOCCAGGIO_TUBO_DX, Stato:=Stato, TimerRisparmio:=TRUE);
  //                 Set_Disp(Ndisp:=BLOCCAGGIO_TUBO_SX, Stato:=Stato, TimerRisparmio:=TRUE);
  //               END_IF;
  //             END_IF;
  //         {
	// 				#endif  //Fine PLAUNO_PLAUNO_LIGHT
  //         }
  //         {
  //         #ifdef TAVOLI_SERPENTINE
  //         }
  //           TAVOLO_POST_ORIZZONTALE:
  //             IF cfg._4RUNNER_TavoliSerpentine=TRUE THEN
  //               IF Disp[Ndisp].statorichiesto<>Disp[Ndisp].stato THEN
  //                 Disp[Ndisp].in_movimento:=TRUE;
  //                 Stato:=LREAL_TO_INT(Disp[Ndisp].statorichiesto);
  //                 //Tavoli posteriori destro e sinistro
  //                 Set_Disp(Ndisp:=TAVOLO_POST_ORIZZ_DX, Stato:=Stato, TimerRisparmio:=TRUE);
  //                 Set_Disp(Ndisp:=TAVOLO_POST_ORIZZ_SX, Stato:=Stato, TimerRisparmio:=TRUE);
  //                 IF (Attesa=TRUE AND i_sys_OPMODE<>AUTOMODE) OR (Attesa=TRUE AND i_sys_OPMODE=AUTOMODE AND TestMasterLavoro()=FALSE) THEN
  //                   WHILE Disp[TAVOLO_POST_ORIZZ_DX].Stato<>Stato OR Disp[TAVOLO_POST_ORIZZ_SX].Stato<>Stato DO
  //                     //Serve per attendere i due tavoli utilizzando la trace del dispositivo fittizzio ma solo se non siamo durante
	// 										//l^esecuzione della tabella stati. In tal caso l^attesa del dispositivo si attende nella prossima riga con flyby a 0
  //                     dret:=_waitTime(T#0ms);
  //                     wait_disp(Device:=TAVOLO_POST_ORIZZONTALE, State:=Stato, Trace:=TRUE);
  //                   END_WHILE;
  //                 END_IF;
  //               END_IF;
  //             END_IF;
  //         {
	// 				#endif  //Fine TAVOLI_SERPENTINE
  //         }
  //         PINZA_ACCOMPAGNAMENTO:
  //           IF Disp[Ndisp].statorichiesto<>Disp[Ndisp].stato THEN
  //             Disp[Ndisp].in_movimento:=TRUE;
  //             CASE Value OF
  //               RIPOSO:
  //                 //Apertura pinza
  //                 Set_Disp(Ndisp:=PINZA_ACCOMPAG_CH_AP, Stato:=RIPOSO, TimerRisparmio:=TRUE);
  //                 IF Attesa=TRUE THEN
  //                   wait_disp(Device:=PINZA_ACCOMPAG_CH_AP,
	// 														State:=RIPOSO,
	// 														Trace:=TRUE);
  //                 END_IF;
  //                 //Arretramento cilindro accompagnamento
  //                 IF Attesa=TRUE THEN
  //                   Set_Disp(Ndisp:=PINZA_ACCOMPAG_AV_IN, Stato:=RIPOSO, TimerRisparmio:=TRUE);
  //                 ELSE
  //                   IF Disp[PINZA_ACCOMPAG_CH_AP].stato=Disp[PINZA_ACCOMPAG_CH_AP].StatoRichiesto THEN
  //                     //In caso di movimento senza attesa, si comanda l^arretramento
  //                     //del carrello di accompagnamento, quando le pinze si sono aperte
  //                     Set_Disp(Ndisp:=PINZA_ACCOMPAG_AV_IN, Stato:=RIPOSO, TimerRisparmio:=TRUE);
  //                   END_IF;
  //                 END_IF;
  //                 IF Attesa=TRUE THEN
  //                   set_trace(Code:=TRC_CARRELLO_ACCOMPAGNAMENTO_INDIETRO);
  //                   wait_disp(Device:=PINZA_ACCOMPAG_AV_IN,
	// 														State:=RIPOSO,
	// 														Trace:=FALSE);
	// 									reset_trace(TRC_CARRELLO_ACCOMPAGNAMENTO_INDIETRO);
  //                 END_IF;
  //               LAVORO:
  //                 //Chiusura pinza
  //                 Set_Disp(Ndisp:=PINZA_ACCOMPAG_CH_AP, Stato:=LAVORO, TimerRisparmio:=TRUE);
  //                 IF Attesa=TRUE THEN
  //                   //Attende se richiesto oppure se la pinza impiega meno di 1 secondo a chiudersi
  //                   wait_disp(Device:=PINZA_ACCOMPAG_CH_AP,
	// 														State:=LAVORO,
	// 														Trace:=FALSE);
  //                   //Avanzamento spintore
  //                   Set_Disp(Ndisp:=PINZA_ACCOMPAG_AV_IN, Stato:=LAVORO, TimerRisparmio:=TRUE);
  //                 ELSE
  //                   IF Disp[PINZA_ACCOMPAG_CH_AP].stato=LAVORO THEN
  //                     //Avanzamento spintore dopo la chiusura pinza, senza attendere per non bloccare
  //                     //il background
  //                     Set_Disp(Ndisp:=PINZA_ACCOMPAG_AV_IN, Stato:=LAVORO, TimerRisparmio:=TRUE);
  //                   END_IF;
  //                 END_IF;
  //               INTERMEDIO:
  //                 //Apertura pinza
  //                 Set_Disp(Ndisp:=PINZA_ACCOMPAG_CH_AP, Stato:=RIPOSO, TimerRisparmio:=TRUE);
  //                 IF Attesa=TRUE THEN
  //                   wait_disp(Device:=PINZA_ACCOMPAG_CH_AP,
	// 														State:=RIPOSO,
	// 														Trace:=FALSE);
  //                 END_IF;
  //             END_CASE;
  //           END_IF;
  //       {
  //       #endif  //Fine FOUR_RUNNER_PLAUNO
  //       }
  //     END_CASE;  //Case dei dispositivi
  //   {
  //   #endif  //Fine RUNNER
  //   }
  // {
  // #else  //Fine ORBITALE
  // }
    //Inizio macchine lineari
    CASE Ndisp OF
      CILSOTTOTESTA:
        IF cfg.SottoTesta3Pos=1 OR cfg.SottoTesta3Pos=2 THEN
          IF Disp[Ndisp].statorichiesto<>Disp[Ndisp].stato THEN
            Disp[Ndisp].in_movimento:=TRUE;
          END_IF;
          CASE TO_INT(Value) OF
            DEVICES_STATUS#RIPOSO:
              IF cfg.SottoTesta3Pos=1 THEN
                //Apertura intermedia cilindro sottotesta
                WriteDigitalOutput(NumOutput:=OUT_CHIUSURA_CILINDRO_SOTTOTESTA, Value:=FALSE);
                WriteDigitalOutput(NumOutput:=OUT_APERTURA_CILINDRO_SOTTOTESTA, Value:=FALSE);
                WriteDigitalOutput(NumOutput:=OUT_APERTURA_INTERMEDIA_CILINDRO_SOTTOTESTA, Value:=TRUE);
              ELSE
                //Apertura totale cilindro sottotesta
                WriteDigitalOutput(NumOutput:=OUT_CHIUSURA_CILINDRO_SOTTOTESTA, Value:=FALSE);
                WriteDigitalOutput(NumOutput:=OUT_APERTURA_CILINDRO_SOTTOTESTA, Value:=TRUE);
                WriteDigitalOutput(NumOutput:=OUT_APERTURA_INTERMEDIA_CILINDRO_SOTTOTESTA, Value:=TRUE);
              END_IF;
              DEVICES_STATUS#LAVORO:
              //Chiusura cilindro sottotesta
              WriteDigitalOutput(NumOutput:=OUT_APERTURA_CILINDRO_SOTTOTESTA, Value:=FALSE);
              WriteDigitalOutput(NumOutput:=OUT_APERTURA_INTERMEDIA_CILINDRO_SOTTOTESTA, Value:=FALSE);
              WriteDigitalOutput(NumOutput:=OUT_CHIUSURA_CILINDRO_SOTTOTESTA, Value:=TRUE);
          END_CASE;
        END_IF;
       SUPPORT_TIRANT:
        // {
        // #ifdef TIRANTE_ANIMA_FC
        // }
        //   IF Disp[Ndisp].statorichiesto<>Disp[Ndisp].stato THEN
        //     Disp[Ndisp].in_movimento:=TRUE;
        //   END_IF;
        //   CASE Value OF
        //     RIPOSO:
        //       Set_Disp(Ndisp:=SOSTEGNO_TIRANTE1, Stato:=RIPOSO, TimerRisparmio:=TRUE);
        //       Set_Disp(Ndisp:=SOSTEGNO_TIRANTE2, Stato:=RIPOSO, TimerRisparmio:=TRUE);
        //     INTERMEDIO:
        //       Set_Disp(Ndisp:=SOSTEGNO_TIRANTE1, Stato:=LAVORO, TimerRisparmio:=TRUE);
        //       Set_Disp(Ndisp:=SOSTEGNO_TIRANTE2, Stato:=RIPOSO, TimerRisparmio:=TRUE);
        //     LAVORO:
        //       Set_Disp(Ndisp:=SOSTEGNO_TIRANTE1, Stato:=LAVORO, TimerRisparmio:=TRUE);
        //       Set_Disp(Ndisp:=SOSTEGNO_TIRANTE2, Stato:=LAVORO, TimerRisparmio:=TRUE);
        //   END_CASE;
        // {
        // #endif  //Fine TIRANTE_ANIMA_FC
        // }
        ;
      // {
      // #ifdef SPINTORE_ULTIMA_CURVA
      // }
      //   SPINTA_ULTIMA_CURVA:
      //     IF Disp[Ndisp].statorichiesto<>Disp[Ndisp].stato THEN
      //       Disp[Ndisp].in_movimento:=TRUE;
      //       CASE Value OF
      //         RIPOSO:
      //           //Spintore indietro e bloccato
      //           Set_Disp(Ndisp:=BLOCCO_SBLOCCO, Stato:=RIPOSO, TimerRisparmio:=TRUE);
      //           wait_disp(Device:=BLOCCO_SBLOCCO, State:=RIPOSO, Trace:=FALSE);
      //           //Arretramento spintore
      //           Set_Disp(Ndisp:=AVANTI_INDIETRO, Stato:=RIPOSO, TimerRisparmio:=TRUE);
      //           wait_disp(Device:=AVANTI_INDIETRO, State:=RIPOSO, Trace:=FALSE);
      //           //Blocco dispositivi di spinta
      //           Set_Disp(Ndisp:=BLOCCO_SBLOCCO, Stato:=LAVORO, TimerRisparmio:=TRUE);
      //           wait_disp(Device:=BLOCCO_SBLOCCO, State:=LAVORO, Trace:=FALSE);
      //         LAVORO:
      //           //Spintore avanti e bloccato
      //           Set_Disp(Ndisp:=BLOCCO_SBLOCCO, Stato:=RIPOSO, TimerRisparmio:=TRUE);
      //           wait_disp(Device:=BLOCCO_SBLOCCO, State:=RIPOSO, Trace:=FALSE);
      //           //Avanzamento spintore
      //           Set_Disp(Ndisp:=AVANTI_INDIETRO, Stato:=LAVORO, TimerRisparmio:=TRUE);
      //           wait_disp(Device:=AVANTI_INDIETRO, State:=LAVORO, Trace:=FALSE);
      //           //Blocco dispositivi di spinta
      //           Set_Disp(Ndisp:=BLOCCO_SBLOCCO, Stato:=LAVORO, TimerRisparmio:=TRUE);
      //           wait_disp(Device:=BLOCCO_SBLOCCO, State:=LAVORO, Trace:=FALSE);
      //         INTERMEDIO:
      //           //Comando di avanzamento spintore senza attesa
      //           Set_Disp(Ndisp:=BLOCCO_SBLOCCO, Stato:=RIPOSO, TimerRisparmio:=TRUE);
      //           wait_disp(Device:=BLOCCO_SBLOCCO, State:=RIPOSO, Trace:=FALSE);
      //           //Avanzamento spintore
      //           Set_Disp(Ndisp:=AVANTI_INDIETRO, Stato:=LAVORO, TimerRisparmio:=TRUE);
      //       END_CASE;
      //     END_IF;
      // // {
      // // #endif  //Fine SPINTORE_ULTIMA_CURVA
      // // }
    END_CASE;
  // {
  // #endif  //Fine macchine lineari
  // }
  ;
END_FUNCTION

FUNCTION_BLOCK FB_PosAsse

  VAR_EXTERNAL
    AssiMaster                      :ARRAY[FIRST_AXIS_MASTER..FIRST_AXIS_MASTER+_CONST_VAR_DEF._MAXAXIS_MASTER#MAXAXIS_MASTER-1] OF MasterAxis;
    Axes                            :ARRAY[_FIRST_AXIS#FIRST_AXIS.._FIRST_AXIS#FIRST_AXIS+_CONST_VAR_DEF._MAXIS#MAXAXIS-1] OF ax;
    UsoPLCOpen						          :BOOL;
  END_VAR

  VAR_EXTERNAL CONSTANT
    FIRST_AXIS_MASTER				      :INT;
  END_VAR

  VAR_INPUT
    Axis                : DB_ANY;
    AttesaResetAxes		  :BOOL;
    //axis              :PosAxis;
    //direction         :EnumDirection;
    positioningMode     :_EnumPositioningMode;
    position          :LREAL;
    //velocityType      :EnumVelocity;
    velocity          :LREAL;
    //positiveAccelType	:EnumAcceleration;
    positiveAccel			:LREAL;
    //negativeAccelType :EnumAcceleration;
    negativeAccel     :LREAL;
    //velocityProfile   :EnumProfile;
    //blendingMode      :EnumBlendingMode;
    //mergeMode         :EnumMergeMode;
    //nextCommand       :EnumNextCommand;
  END_VAR
  VAR
    dret							:DINT;
		axisInt						:INT;
		//thisCommand				:commandIDType;

		CURRENT_STATE			:INT:=GENERAL_STATE#STATE_INIT;
		AttesaFineResetAssi:FB_AttesaFineResetAssi;
  END_VAR
	VAR_OUTPUT
		OutputState:INT;
	END_VAR
	CASE CURRENT_STATE OF
		GENERAL_STATE#STATE_INIT:
			IF AttesaResetAxes=TRUE THEN
				IF (AttesaFineResetAssi.outputState<>GENERAL_STATE#STATE_END) THEN
					AttesaFineResetAssi();
				ELSE
					AttesaFineResetAssi();
					IF (UsoPLCOpen) THEN
						CURRENT_STATE:=_FB_PosAsse#STATE_POSASSE_PLCOPEN;
					ELSE
						//thisCommand:=_getCommandID();
						CURRENT_STATe:=_FB_PosAsse#STATE_POSASSE_NOPLCOPEN;
					END_IF;
				END_IF;
			ELSE
				IF (UsoPLCOpen) THEN
					CURRENT_STATE:=_FB_PosAsse#STATE_POSASSE_PLCOPEN;
				ELSE
					//thisCommand:=_getCommandID();
					CURRENT_STATe:=_FB_PosAsse#STATE_POSASSE_NOPLCOPEN;
				END_IF;
			END_IF;

      _FB_PosAsse#STATE_POSASSE_PLCOPEN:
			axisInt:=GetAxisFromTO(axis);
      IF positioningMode = _EnumPositioningMode#ABSOLUTE THEN

        IF (axisInt=-1) THEN
          axisInt:=GetMasterAxisFromTO(axis);
          AssiMaster[axisInt].MC_Axes.move_abs_param.Position :=position;
          AssiMaster[axisInt].MC_Axes.move_abs_param.Velocity:=velocity;
          AssiMaster[axisInt].MC_Axes.move_abs_param.Acceleration:=positiveAccel;
          AssiMaster[axisInt].MC_Axes.move_abs_param.Deceleration:=negativeAccel;
          AssiMaster[axisInt].MC_Axes.move_absolute := TRUE ;
        ELSE
          Axes[axisInt].MC_Axes.move_abs_param.Position :=position;
          Axes[axisInt].MC_Axes.move_abs_param.Velocity:=velocity;
          Axes[axisInt].MC_Axes.move_abs_param.Acceleration:=positiveAccel;
          Axes[axisInt].MC_Axes.move_abs_param.Deceleration:=negativeAccel;
          Axes[axisInt].MC_Axes.move_absolute := TRUE ;
        END_IF;

    ELSE
        IF (axisInt=-1) THEN
          axisInt:=GetMasterAxisFromTO(axis);
          AssiMaster[axisInt].MC_Axes.move_rel_param.Distance :=position;
          AssiMaster[axisInt].MC_Axes.move_rel_param.Velocity:=velocity;
          AssiMaster[axisInt].MC_Axes.move_rel_param.Acceleration:=positiveAccel;
          AssiMaster[axisInt].MC_Axes.move_rel_param.Deceleration:=negativeAccel;
          AssiMaster[axisInt].MC_Axes.move_relative:=TRUE;
        ELSE
          Axes[axisInt].MC_Axes.move_rel_param.Distance :=position;
          Axes[axisInt].MC_Axes.move_rel_param.Velocity:=velocity;
          Axes[axisInt].MC_Axes.move_rel_param.Acceleration:=positiveAccel;
          Axes[axisInt].MC_Axes.move_rel_param.Deceleration :=negativeAccel;
          Axes[axisInt].MC_Axes.move_relative:=TRUE;
        END_IF;
    END_IF;

			CURRENT_STATE:=GENERAL_STATE#STATE_END;

		_FB_PosAsse#STATE_POSASSE_NOPLCOPEN:

			(*dret:=_pos(axis:=axis,
								 direction:=direction,
								 positioningMode:=positioningMode,
								 position:=position,
								 velocityType:=velocityType,
								 velocity:=velocity,
								 positiveAccelType:=positiveAccelType,
								 positiveAccel:=positiveAccel,
								 negativeAccelType:=DIRECT,
								 negativeAccel:=negativeAccel,
								 velocityProfile:=velocityProfile,
								 blendingMode:=blendingMode,
								 mergeMode:=mergeMode,
								 nextCommand:=IMMEDIATELY,
								 commandId:=thisCommand);*)
			// IF (nextCommand=IMMEDIATELY) THEN
			// 	CURRENT_STATE:=GENERAL_STATE#STATE_END;
			// ELSE
			// 	IF NOT (dret=7001 OR dret=7002) THEN
					CURRENT_STATE:=GENERAL_STATE#STATE_END;
			// 	END_IF;
			// END_IF;

		GENERAL_STATE#STATE_END:
			CURRENT_STATE:=GENERAL_STATE#STATE_INIT;
	END_CASE;
	OutputState:=CURRENT_STATE;
END_FUNCTION_BLOCK

/****************************************************************
 * WAITS UNTIL THERE IS NO LONGER ANY RESET COMMAND ON ALL AXES *
 ****************************************************************/

FUNCTION_BLOCK FB_AttesaFineResetAssi

  VAR_EXTERNAL
    Axes                            :ARRAY[_FIRST_AXIS#FIRST_AXIS.._FIRST_AXIS#FIRST_AXIS+_CONST_VAR_DEF._MAXIS#MAXAXIS-1] OF ax;
    pm                              : ARRAY[_FIRST_AXIS#FIRST_AXIS.._FIRST_AXIS#FIRST_AXIS+_CONST_VAR_DEF._MAXIS#MAXAXIS-1] OF AxisParameters;
  END_VAR

  VAR_EXTERNAL CONSTANT
    TRC_WAIT_FOR_DRIVE_COMMUNICATION    :INT;
  END_VAR

  VAR
    posax : REF_TO TO_SynchronousAxis;
    i      :INT;
    dret  :DINT;

		CURRENT_STATE:INT:=GENERAL_STATE#STATE_INIT;
		CURRENT_AXIS:INT;
  END_VAR

	VAR_OUTPUT
		OutputState:INT;
	END_VAR

	CASE CURRENT_STATE OF
		GENERAL_STATE#STATE_INIT:
			CURRENT_AXIS:=_FIRST_AXIS#FIRST_AXIS-1;
			CURRENT_STATE:=_FB_AttesaFineResetAssi#STATE_ATTESA_FINE_RESET_ASSI_CICLO_ASSI;

      _FB_AttesaFineResetAssi#STATE_ATTESA_FINE_RESET_ASSI_CICLO_ASSI:
			CURRENT_AXIS:=CURRENT_AXIS+1;
			IF CURRENT_AXIS<_MAXIS#MAXAXIS THEN
				IF pm[CURRENT_AXIS].ma_asse_abilitato=TRUE THEN
					CURRENT_STATE:=_FB_AttesaFineResetAssi#STATE_WAIT_ATTESA_AZIONAMENTO;
				END_IF;
			ELSE
				CURRENT_AXIS:=_FIRST_AXIS#FIRST_AXIS-1;
				CURRENT_STATE:=GENERAL_STATE#STATE_END;
			END_IF;

      _FB_AttesaFineResetAssi#STATE_WAIT_ATTESA_AZIONAMENTO:
			posax := AsSynchronousAxisRef(Axes[CURRENT_AXIS].posax);
      IF posax^.StatusWord.%X2 THEN
				set_trace(Code:=TRC_WAIT_FOR_DRIVE_COMMUNICATION, Axis:=CURRENT_AXIS);
			ELSE
				reset_trace(Code:=TRC_WAIT_FOR_DRIVE_COMMUNICATION);
				CURRENT_STATE:=_FB_AttesaFineResetAssi#STATE_ATTESA_FINE_RESET_ASSI_CICLO_ASSI;
			END_IF;

		GENERAL_STATE#STATE_END:
			CURRENT_STATE:=GENERAL_STATE#STATE_INIT;
	END_CASE;
	OutputState:=CURRENT_STATE;
END_FUNCTION_BLOCK

FUNCTION GetAxisFromTO:INT

  VAR_EXTERNAL
    Axes                            :ARRAY[_FIRST_AXIS#FIRST_AXIS.._FIRST_AXIS#FIRST_AXIS+_CONST_VAR_DEF._MAXIS#MAXAXIS-1] OF ax;
  END_VAR

	VAR_INPUT
		Axis	: DB_ANY;
	END_VAR

	VAR
		i			:INT;
   posax : REF_TO TO_SynchronousAxis;
   LocAxis : REF_TO TO_SynchronousAxis;
	END_VAR

	GetAxisFromTO:=-1;
  LocAxis := AsSynchronousAxisRef(Axis);

	FOR i:=0 TO _MAXIS#MAXAXIS -1 DO
  posax:= AsSynchronousAxisRef(Axes[i].PosAx);
    IF (PosAx=LocAxis) THEN
		//IF (Axes[i].PosAx=Axis) THEN
			GetAxisFromTO:=i;
		END_IF;
	END_FOR;
END_FUNCTION

END_NAMESPACE
